Yaskawa INFORM job: X2_34-37(-90,0).JBI

/JOB
//NAME X2_34-37(-90,0)
//POS
///NPOS 478,478,478,11,0,0
///TOOL 0
///POSTYPE PULSE
///PULSE
C00000=59350,-53311,-57323,3430,41392,19515
C00001=122728,-72765,-37270,-45372,18157,11336
C00002=113002,-9355,-31874,-9491,78881,-10162
C00003=107008,40287,15446,-7646,74688,-11911
C00004=107149,45804,24218,-7788,72161,-11701
C00005=108392,48192,28010,-10243,72680,-1076
C00006=108392,48392,29954,-10302,71604,-983
C00007=108392,48331,29423,-10286,71896,-1009
C00008=108010,50265,31522,-10186,71551,-1114
C00009=108392,48331,29423,-10286,71896,-1009
C00010=108911,49901,30550,-10443,72076,-8021
C00011=109414,51873,32709,-10619,71831,-7821
C00012=108911,49901,30550,-10443,72076,-8021
C00013=102203,43615,23227,-8248,72569,-10434
C00014=106081,49085,29485,-15378,74997,-2308
C00015=106081,49206,30588,-15419,74401,-2232
C00016=106081,49153,30130,-15402,74647,-2263
C00017=105730,50968,32108,-15326,74307,-2347
C00018=106081,49153,30130,-15402,74647,-2263
C00019=108167,43461,21271,-12324,74506,-6920
C00020=107374,42085,15448,-7738,75637,-11845
C00021=120191,30165,1303,-6226,81332,6626
C00022=119709,34887,8992,-6124,79003,6581
C00023=119523,36874,12198,-6088,78043,6565
C00024=119519,36825,13807,-6108,77033,6613
C00025=119523,36874,12198,-6088,78043,6565
C00026=119515,36764,13496,-6103,77191,6604
C00027=119868,39633,16467,-6214,76866,6741
C00028=119515,36764,13496,-6103,77191,6604
C00029=121889,32783,9008,-6775,78090,7366
C00030=122776,40716,17165,-7052,77228,7717
C00031=121823,41691,18182,-6780,77023,7402
C00032=122776,40716,17165,-7052,77228,7717
C00033=121889,32783,9008,-6775,78090,7366
C00034=119523,36874,12198,-6088,78043,6565
C00035=119709,34887,8992,-6124,79003,6581
C00036=120191,30165,1303,-6226,81332,6626
C00037=121604,30205,1144,-6630,81559,7083
C00038=121089,34887,8794,-6520,79231,7034
C00039=120890,36858,11983,-6481,78271,7017
C00040=120886,36803,13585,-6502,77262,7069
C00041=120890,36858,11983,-6481,78271,7017
C00042=120878,36774,13282,-6496,77432,7057
C00043=121214,39658,16269,-6601,77105,7189
C00044=120878,36774,13282,-6496,77432,7057
C00045=120486,37076,13561,-6383,77385,6926
C00046=119528,38122,14634,-6107,77190,6608
C00047=120486,37076,13561,-6383,77385,6926
C00048=120682,35058,10322,-6419,78351,6942
C00049=121186,30266,2562,-6523,80690,6990
C00050=134026,40869,15057,4047,52311,47824
C00051=133273,45805,23219,4742,49872,47398
C00052=132981,47914,26662,5033,48858,47219
C00053=132978,48047,28467,5116,47820,47163
C00054=132981,47914,26662,5033,48858,47219
C00055=130421,47335,28194,14259,47961,42182
C00056=130639,50701,31849,14213,47420,42201
C00057=132969,48064,28169,5108,48012,47169
C00058=135543,46606,26609,3148,48091,48321
C00059=135868,54135,34684,2953,46980,48432
C00060=134925,54643,35244,3684,46935,48001
C00061=135868,54135,34684,2953,46980,48432
C00062=135543,46606,26609,3148,48091,48321
C00063=132981,47914,26662,5033,48858,47219
C00064=133273,45805,23219,4742,49872,47398
C00065=134026,40869,15057,4047,52311,47824
C00066=158164,35728,9631,-12841,54320,57618
C00067=156933,39530,16487,-12369,51918,57402
C00068=156452,41160,19364,-12190,50934,57317
C00069=156450,41229,21096,-12367,49926,57444
C00070=156452,41160,19364,-12190,50934,57317
C00071=156479,41102,20610,-12346,50159,57426
C00072=156356,44237,23924,-12335,49721,57428
C00073=156479,41102,20610,-12346,50159,57426
C00074=155785,40986,20547,-11858,50036,57137
C00075=154785,40646,20189,-11137,49940,56708
C00076=155785,40986,20547,-11858,50036,57137
C00077=156262,39303,17617,-12037,51024,57224
C00078=157483,35375,10637,-12509,53434,57446
C00079=160593,39475,13550,-14508,54241,58615
C00080=159342,43270,20469,-14089,51785,58436
C00081=158853,44905,23381,-13934,50776,58367
C00082=158852,45007,25149,-14138,49770,58512
C00083=158853,44905,23381,-13934,50776,58367
C00084=155515,42876,22536,-2607,48655,51694
C00085=155529,45453,25272,-2635,48295,51710
C00086=158854,44932,24718,-14094,49990,58481
C00087=161444,46441,26342,-15939,50249,59595
C00088=161040,53766,34331,-15923,49060,59612
C00089=160097,53171,33669,-15238,48978,59196
C00090=161040,53766,34331,-15923,49060,59612
C00091=161444,46441,26342,-15939,50249,59595
C00092=158853,44905,23381,-13934,50776,58367
C00093=159342,43270,20469,-14089,51785,58436
C00094=160593,39475,13550,-14508,54241,58615
C00095=148971,42504,16746,-4915,52183,53021
C00096=147979,47046,24523,-4355,49683,52716
C00097=147593,48996,27807,-4132,48646,52593
C00098=147590,49137,29621,-4197,47605,52637
C00099=147593,48996,27807,-4132,48646,52593
C00100=148206,49324,28699,-4616,48299,52880
C00101=148386,52346,32006,-4787,47830,52984
C00102=147610,49163,29309,-4198,47810,52637
C00103=147454,49128,29272,-4080,47808,52567
C00104=147457,49325,29466,-4083,47790,52569
C00105=146486,49526,29681,-3347,47716,52137
C00106=147457,49325,29466,-4083,47790,52569
C00107=147454,49128,29272,-4080,47808,52567
C00108=147593,48996,27807,-4132,48646,52593
C00109=147979,47046,24523,-4355,49683,52716
C00110=148753,37651,9035,-4624,54413,52827
C00111=162629,67371,16666,-14387,95994,52782
C00112=162715,57365,2812,-16324,103951,51832
C00113=160874,53905,-839,-17120,106140,50911
C00114=173545,40340,-5560,-32046,95660,52318
C00115=172356,48440,2674,-29251,92100,53433
C00116=172375,50726,4522,-29031,92137,53493
C00117=171941,50016,3368,-28017,91820,53556
C00118=172934,47472,3029,-30290,87254,54349
C00119=166298,46940,-5204,-15814,93409,53604
C00120=167727,47900,-7727,-16302,95626,53755
C00121=154370,-11928,-49618,9666,90717,31299
C00122=126601,-55902,-47749,13735,83134,-9694
C00123=110572,-56965,-55890,14658,90278,-14468
C00124=134387,-39172,-38807,-12376,86277,20344
C00125=136266,-41846,-34601,-16059,78566,27361
C00126=135831,-39745,-32201,-16023,78101,27269
C00127=132382,-45209,-35546,-15612,76705,26216
C00128=133414,-53213,-38184,-18925,70500,23054
C00129=132483,-55031,-38922,-19056,69495,22520
C00130=133928,-49591,-35946,-21097,73532,26608
C00131=127522,-56914,-39892,-20235,70668,24713
C00132=130575,-58808,-42172,-20683,71834,25657
C00133=131419,-52897,-41760,-13173,72105,2236
C00134=151757,-37235,-32664,-25855,92713,16023
C00135=148694,-31120,-30848,-28555,97484,16481
C00136=152363,20888,-11521,-23566,108052,25705
C00137=155491,63274,13853,-18429,111086,34801
C00138=150514,89045,46229,-21307,107758,32982
C00139=149106,88504,48693,-21100,105732,32842
C00140=153713,50743,12699,-33613,93756,12076
C00141=152514,62453,23514,-30409,96198,11306
C00142=153571,72354,35346,-30285,92331,9677
C00143=151039,57679,18624,-26133,86933,-1110
C00144=146574,45095,4989,-17377,80841,-11651
C00145=146416,46512,5286,-14277,82040,-14909
C00146=141388,39329,-953,-2943,76634,-26635
C00147=140619,46287,2526,-1728,82676,-28626
C00148=139837,43342,-3801,-1439,85041,-28899
C00149=141798,27002,-27786,-2149,91441,-28405
C00150=143772,-19107,-38740,-14355,94017,12677
C00151=143698,-35148,-33847,-20276,92427,33189
C00152=141918,-24797,-26817,-20326,92921,32464
C00153=139594,-23350,-22642,-20301,90627,32011
C00154=140500,-47178,-33366,-23894,71804,30939
C00155=143725,-38410,-27629,-28409,78422,12628
C00156=143636,-41247,-28872,-28024,73501,10134
C00157=137881,-52583,-35183,-23334,62436,-881
C00158=129248,-60396,-38780,-13341,52739,-14402
C00159=124267,-62494,-40095,-3055,50610,-24451
C00160=119084,-58248,-39599,7242,55598,-36917
C00161=117935,-60108,-42034,7672,56240,-37337
C00162=115664,-65010,-47736,8512,57449,-38158
C00163=121785,-61828,-52329,5505,69210,-35118
C00164=148930,-33628,-41038,-4538,77484,-18447
C00165=163858,24222,1645,-10794,81228,-7547
C00166=163712,28964,9442,-10824,78886,-7392
C00167=163375,31110,12798,-10770,77896,-7422
C00168=162966,25989,8902,-6453,74358,251
C00169=171220,35624,19743,-19386,77626,18928
C00170=174903,69588,56637,-24731,86432,36485
C00171=176281,62245,51753,-30189,71814,61901
C00172=174700,53660,39403,-25265,70725,61619
C00173=176244,52382,34806,-25393,73168,61673
C00174=174832,57379,31343,-14926,87681,59388
C00175=147451,1111,-29714,-5377,100632,19781
C00176=112791,-31989,-50015,2241,90212,-24459
C00177=107981,-35875,-46971,4517,78040,-26268
C00178=109410,-31915,-41181,4141,76439,-25836
C00179=109643,-29612,-38300,4087,75838,-25775
C00180=108775,-25319,-36143,8282,81258,-19579
C00181=113815,-28658,-38499,3030,79667,-8408
C00182=120146,-28725,-38561,-4150,79807,1674
C00183=136607,-12516,-23650,-24736,88445,21917
C00184=138997,-10914,-21244,-25939,84896,23287
C00185=136597,-19153,-27062,-20495,74929,32505
C00186=127631,-24253,-35023,-5775,74490,30240
C00187=129181,-27934,-40726,-6212,76213,30690
C00188=139651,-3107,-33687,-4364,86662,-15844
C00189=140099,618,-27389,-4493,84729,-15631
C00190=139833,2398,-24483,-4425,83841,-15689
C00191=138545,5945,-22338,1327,87046,-9478
C00192=148216,2445,-23282,-11424,83992,10224
C00193=153040,10099,-16158,-17812,86817,20381
C00194=156294,19571,-6705,-22682,89726,28901
C00195=159272,37595,11787,-27323,93895,28698
C00196=154169,16276,-8816,-16740,78788,38767
C00197=152712,20066,-9195,-12847,84122,38020
C00198=154297,18366,-13942,-13242,86364,38311
C00199=143466,6998,19042,-5158,32162,41222
C00200=147237,-51968,-50099,4175,73083,42408
C00201=-3643,-76224,-106676,-19950,71810,-76872
C00202=-6047,-95755,-92046,14751,98253,-9605
C00203=-2299,-70459,-84112,3705,91093,-18065
C00204=-2299,-70459,-84112,3705,91093,-18065
C00205=-2299,-70459,-84112,3705,91093,-18065
C00206=-2299,-70459,-84112,3705,91093,-18065
C00207=61951,-108908,-90353,7974,21769,-53190
C00208=44975,-75191,-76287,54105,62461,-71292
C00209=78581,-58710,-61930,31634,35162,-55381
C00210=94816,-22771,-39143,38147,43253,-85351
C00211=95668,-20492,-32997,40754,37729,-87628
C00212=95668,-20442,-31356,41600,36978,-88107
C00213=95668,-20481,-32513,41001,37505,-87770
C00214=95495,-18068,-30743,41020,37699,-87770
C00215=95668,-20481,-32513,41001,37505,-87770
C00216=89708,-21268,-34265,45191,40885,-89740
C00217=90261,-15540,-28471,45297,40161,-89843
C00218=90261,-15513,-27582,45749,39780,-90110
C00219=90261,-15527,-28007,45532,39961,-89983
C00220=91375,-15045,-27644,44668,39419,-89560
C00221=90261,-15527,-28007,45532,39961,-89983
C00222=88067,4046,-12693,46606,41526,-90451
C00223=88067,4066,-11724,47089,41117,-90741
C00224=88067,4053,-12277,46812,41349,-90575
C00225=89178,4455,-11933,46018,40776,-90188
C00226=88067,4046,-12908,46498,41617,-90387
C00227=93864,-1171,-17172,27469,32670,-81316
C00228=93864,-1150,-16127,27931,32107,-81561
C00229=93864,-1161,-16600,27720,32361,-81450
C00230=93686,724,-15030,27925,32421,-81546
C00231=93864,-1171,-17458,27343,32827,-81250
C00232=86880,-2670,-19039,34652,35541,-84684
C00233=77447,40941,12142,46518,66528,-79108
C00234=77447,40828,13235,46743,66015,-79371
C00235=77447,40915,12396,46570,66408,-79170
C00236=78189,41279,12776,46293,66002,-79003
C00237=77447,40915,12396,46570,66408,-79170
C00238=77711,61383,34518,44784,60703,-78470
C00239=77711,61401,35861,45103,60114,-78770
C00240=77711,61383,34367,44748,60769,-78437
C00241=78627,62334,35456,44423,60182,-78251
C00242=77711,61383,34367,44748,60769,-78437
C00243=87327,38488,-37,11684,57539,-57739
C00244=92703,33891,441,-7168,52274,-42102
C00245=94252,42993,11540,-8600,52099,-41498
C00246=94252,42798,12742,-8697,51267,-41425
C00247=94252,42977,11640,-8607,52029,-41490
C00248=94205,45159,13958,-8608,51725,-41483
C00249=94252,42977,11640,-8607,52029,-41490
C00250=88553,40317,7447,-4237,52798,-43866
C00251=77780,64504,35767,30085,55551,-63063
C00252=77882,64751,36053,30043,55472,-63041
C00253=77882,64734,37138,30274,54883,-63228
C00254=77882,64751,36157,30064,55416,-63059
C00255=78504,65403,36908,29747,55085,-62879
C00256=77882,64751,36157,30064,55416,-63059
C00257=77930,65478,35918,25842,53172,-64425
C00258=75957,78225,52136,32216,53612,-64557
C00259=75957,78336,53316,32477,53042,-64758
C00260=75957,78231,52217,32233,53572,-64572
C00261=76543,78457,52489,31920,53306,-64380
C00262=75957,78231,52217,32233,53572,-64572
C00263=75783,52857,14963,26033,68951,-61065
C00264=76778,51540,16645,25850,67104,-61119
C00265=76553,54259,19675,26040,66751,-61289
C00266=76152,68337,35819,26754,64443,-62008
C00267=76309,68979,36633,26729,64087,-61973
C00268=76161,73805,46213,28343,55084,-61966
C00269=76040,75497,47702,28425,55082,-62022
C00270=75485,77195,52229,31394,50715,-63899
C00271=76358,61277,29656,23751,52989,-59172
C00272=75244,23807,-9833,23130,57943,-58480
C00273=78328,30150,-3634,21247,56637,-57509
C00274=82524,40429,3879,10756,62616,-55403
C00275=83243,40821,5102,10290,61963,-55146
C00276=92066,29463,-1741,-9440,53850,-44784
C00277=92409,29931,-1279,-9693,53846,-44645
C00278=95822,30058,-1154,-12140,54276,-43316
C00279=92072,29548,-1666,-1163,53131,-49252
C00280=90114,17633,-16179,284,55928,-50028
C00281=80680,14818,-24193,20442,65844,-59872
C00282=77180,38928,7111,43331,74666,-71993
C00283=76673,54469,24090,43953,73098,-72919
C00284=76771,55672,25429,43962,72900,-72963
C00285=76784,55849,25626,43964,72871,-72969
C00286=78172,63512,34338,39520,65661,-69940
C00287=79648,59091,29288,35397,62522,-67074
C00288=75980,37060,-454,35377,69732,-66149
C00289=81483,21043,-13915,32107,67437,-64274
C00290=93507,15990,-19907,5211,64480,-50669
C00291=99800,11020,-22513,-5623,60000,-50039
C00292=99783,5101,-23986,-5176,53212,-49502
C00293=100096,6075,-23185,433,53012,-52451
C00294=100559,6099,-23054,81,52942,-52266
C00295=100559,6099,-23054,81,52942,-52266
C00296=95780,-7481,-38206,3595,55393,-54089
C00297=86068,-7258,-38029,32714,65078,-69570
C00298=89977,-5445,-32844,31222,61873,-68759
C00299=89643,-3500,-31211,31407,61985,-68864
C00300=88246,9256,-20330,32202,62368,-69333
C00301=88278,10099,-19644,32183,62365,-69319
C00302=87437,19709,-10754,32777,62224,-69720
C00303=93562,10508,-19170,18010,55559,-61503
C00304=91617,5056,-25544,19093,57043,-62018
C00305=90732,-18366,-45622,16723,54511,-62954
C00306=99990,-18392,-38429,13920,44377,-71620
C00307=100837,-18665,-38703,13148,44269,-71234
C00308=97918,-19792,-36092,25968,40989,-77255
C00309=98001,-23338,-34358,32939,34367,-85184
C00310=99551,-14617,-34520,26965,45535,-82533
C00311=93873,-14551,-28302,47146,43784,-90863
C00312=93873,-14551,-28302,47146,43784,-90863
C00313=92894,-25654,-38538,40707,40207,-87648
C00314=51114,-81290,-74278,61960,52593,-60278
C00315=6076,-109546,-85200,71251,79672,-70600
C00316=6076,-109546,-85200,71251,79672,-70600
C00317=6076,-109546,-85200,-4239,76823,-70600
C00318=-8024,-164446,-133802,16041,6272,-12396
C00319=-8024,-164446,-133802,16041,6272,-12396
C00320=-80911,-131071,-112390,19160,57527,4768
C00321=-107387,-112645,-89313,18613,48039,3448
C00322=-120529,-94925,-67119,18087,38914,2179
C00323=-102807,-11704,-32462,5874,76695,13415
C00324=-103436,-3791,-23255,6127,75148,13126
C00325=-103560,-1765,-20423,6188,74460,13051
C00326=-103560,-1806,-19122,6212,73642,13010
C00327=-103601,-1431,-19452,6214,74041,13015
C00328=-104452,277,-18031,6506,74110,12725
C00329=-103539,-2063,-20212,6189,74177,13043
C00330=-120126,-10436,-31938,6011,80471,-6680
C00331=-119034,-8056,-29018,5697,79822,-6345
C00332=-119034,-8150,-28117,5707,79221,-6375
C00333=-119034,-8056,-29018,5697,79822,-6345
C00334=-118636,-7203,-28340,5579,79816,-6211
C00335=-119064,-5644,-27091,5704,79877,-6351
C00336=-118636,-7203,-28340,5579,79816,-6211
C00337=-122253,-9472,-30321,6643,80135,-7408
C00338=-122707,-3013,-24427,6779,79866,-7571
C00339=-122021,-2022,-23613,6578,79819,-7343
C00340=-122707,-3013,-24427,6779,79866,-7571
C00341=-121204,9301,-16198,6319,81003,-7011
C00342=-120979,11415,-12534,6272,79823,-6996
C00343=-120979,11346,-11871,6278,79382,-7018
C00344=-120979,11415,-12534,6272,79823,-6996
C00345=-121673,13624,-10544,6477,79786,-7230
C00346=-120979,11415,-12534,6272,79823,-6996
C00347=-121039,12182,-11846,8037,80321,-9006
C00348=-120294,13253,-10880,7825,80206,-8763
C00349=-121039,12182,-11846,8037,80321,-9006
C00350=-121310,5674,-20943,6336,82061,-6993
C00351=-139815,-25323,-43479,19,53677,-50237
C00352=-137572,-18164,-33682,-1617,51348,-49297
C00353=-137572,-18186,-32944,-1627,50884,-49290
C00354=-137572,-18164,-33682,-1617,51348,-49297
C00355=-138000,-16627,-32540,-1306,51428,-49477
C00356=-137572,-18164,-33682,-1617,51348,-49297
C00357=-141541,-18207,-34048,1274,51544,-50959
C00358=-141186,-12326,-28968,1018,51433,-50811
C00359=-140737,-11536,-28358,690,51458,-50623
C00360=-141186,-12326,-28968,1018,51433,-50811
C00361=-159686,26179,2441,14066,53601,-58348
C00362=-159232,27229,5186,13963,52408,-58323
C00363=-159232,27222,5932,14048,51958,-58386
C00364=-159232,27229,5186,13963,52408,-58323
C00365=-159232,27225,5485,13997,52227,-58349
C00366=-159220,29212,7438,14024,52052,-58369
C00367=-159232,27225,5485,13997,52227,-58349
C00368=-164735,35698,13654,29808,58437,-68077
C00369=-164028,35618,13572,29436,58200,-67836
C00370=-164735,35698,13654,29808,58437,-68077
C00371=-161795,29787,7764,15728,52595,-59373
C00372=-161795,29788,8601,15834,52098,-59452
C00373=-161795,29787,7764,15728,52595,-59373
C00374=-161783,31729,9695,15761,52409,-59396
C00375=-161795,29787,7764,15728,52595,-59373
C00376=-165243,28841,7606,18106,52930,-60800
C00377=-165806,38731,16984,22046,53706,-63214
C00378=-165192,38605,16853,21659,53559,-62976
C00379=-165806,38731,16984,22046,53706,-63214
C00380=-161708,46386,23154,8907,61269,-44547
C00381=-161224,48066,26131,8737,60259,-44442
C00382=-161222,48202,27939,8826,59228,-44523
C00383=-161224,48066,26131,8737,60259,-44442
C00384=-161238,48238,27638,8816,59431,-44513
C00385=-161118,51495,31180,8798,58918,-44508
C00386=-161238,48238,27638,8816,59431,-44513
C00387=-161086,48113,27502,8735,59433,-44454
C00388=-161078,48307,27691,8732,59416,-44452
C00389=-160108,47930,27281,8216,59373,-44078
C00390=-161078,48307,27691,8732,59416,-44452
C00391=-161086,48113,27502,8735,59433,-44454
C00392=-161224,48066,26131,8737,60259,-44442
C00393=-161708,46386,23154,8907,61269,-44547
C00394=-162944,42495,16096,9351,63722,-44812
C00395=-174609,85782,55206,18480,94121,-57514
C00396=-173388,84153,56528,18357,92279,-57362
C00397=-178295,72858,49572,29598,87914,-53870
C00398=-178363,71681,49458,30316,81279,-55416
C00399=-178775,74747,53745,31442,79609,-55982
C00400=-178120,80280,53499,25679,87195,-54196
C00401=-177788,66292,45128,22799,80541,-57078
C00402=-165876,20944,-7359,14016,91072,-47752
C00403=-144031,-8096,-47002,-481,102749,-33013
C00404=-113249,-55125,-55779,-6617,87879,14622
C00405=-105402,-49476,-43093,-17129,78821,17705
C00406=-107372,-45114,-37354,-16923,77172,17229
C00407=-107897,-43226,-34630,-16890,76385,17150
C00408=-123036,-54169,-41018,3647,66196,9526
C00409=-125103,-54109,-40569,7539,65613,9158
C00410=-133018,-52183,-38196,18552,67287,3963
C00411=-135096,-56008,-41994,19101,68310,3149
C00412=-148619,-36280,-33179,26254,90102,-11601
C00413=-132022,-46525,-51369,8915,93592,-12104
C00414=-152394,4325,-31091,21424,100011,-27739
C00415=-150620,74441,30669,21497,109248,-32750
C00416=-152126,53419,9650,25324,101365,-34081
C00417=-152823,56464,14992,29675,98105,-11003
C00418=-153512,66710,26766,28901,94570,-8735
C00419=-151176,53481,12027,24882,88967,903
C00420=-148217,46273,4019,19056,85273,8690
C00421=-145575,40234,-2364,10924,81880,17637
C00422=-142774,42237,-1321,4504,82417,25550
C00423=-141310,41249,-3509,1904,83312,28397
C00424=-140520,38377,-9680,1608,85617,28672
C00425=-145482,-30493,-50756,14636,95383,-13188
C00426=-142176,-26033,-28146,20229,92686,-32606
C00427=-139838,-24569,-23969,20194,90398,-32145
C00428=-141333,-43488,-32424,24355,75177,-35516
C00429=-142946,-39788,-29545,27566,77515,-12382
C00430=-142712,-38988,-29426,26650,76094,-9122
C00431=-137490,-51139,-36024,22440,64589,1384
C00432=-129219,-61272,-40095,12800,52551,14455
C00433=-125098,-62268,-41395,3949,52110,22670
C00434=-120434,-59895,-41306,-5152,54802,34175
C00435=-118218,-60267,-42467,-7826,55944,37248
C00436=-115940,-65207,-48159,-8687,57132,38075
C00437=-158051,-33814,-49892,7441,80913,13725
C00438=-163513,25616,3177,10792,80459,7597
C00439=-163372,30455,11081,10830,78103,7439
C00440=-163993,28142,11085,12803,74423,6981
C00441=-161648,29238,11147,4496,75447,179
C00442=-171143,45412,28292,19077,81279,-23270
C00443=-173705,65046,50293,22854,85176,-36170
C00444=-173974,62485,49606,24076,73199,-49227
C00445=-172570,70781,55370,19160,78152,-47867
C00446=-174025,68948,50025,19270,80716,-47984
C00447=-170072,38309,9009,5458,81396,-48416
C00448=-145937,-33300,-50613,2555,87892,-10434
C00449=-117969,-26674,-50251,-1455,96093,22658
C00450=-108065,-36096,-47601,-4778,77881,26213
C00451=-109507,-32110,-41823,-4391,76297,25779
C00452=-109013,-37865,-42571,-5415,69231,26193
C00453=-107679,-33877,-40967,-9851,74714,20356
C00454=-113110,-32097,-41032,-3661,77261,8676
C00455=-119719,-29513,-40298,3828,79988,-1546
C00456=-130402,-22376,-34110,15555,82843,-20591
C00457=-132503,-6978,-23545,15597,88653,-21115
C00458=-133170,-4219,-21374,15691,88857,-21320
C00459=-127848,-25408,-36231,5685,74178,-30350
C00460=-129407,-29126,-41925,6135,75876,-30806
C00461=-139811,-3516,-34603,4319,86523,15767
C00462=-140259,233,-28314,4452,84609,15556
C00463=-139695,2013,-26001,4296,84073,15716
C00464=-138357,5152,-24179,-1260,87195,9766
C00465=-142581,5884,-23661,3711,87904,-1101
C00466=-150814,13438,-16434,14780,91136,-16214
C00467=-153585,30594,-714,18230,97958,-27100
C00468=-154794,42503,11376,18274,96962,-27667
C00469=-154809,42525,11398,18275,96963,-27672
C00470=-153093,18834,-10833,12947,84050,-38162
C00471=-154693,17143,-15552,13354,86281,-38457
C00472=-149017,-30265,-44675,21897,62232,-30468
C00473=-102406,-109115,-77602,2898,35707,11807
C00474=-80911,-131071,-112390,19160,57527,4768
C00475=-8024,-164446,-133802,16041,6272,-12396
C00476=-8024,-164446,-133802,16041,6272,-12396
C00477=6076,-109546,-85200,-4239,76823,-70600
BC00000=228604,517006,641220
BC00001=287751,517515,392862
BC00002=287751,487719,199707
BC00003=287751,487719,199707
BC00004=287751,487719,199707
BC00005=287751,487719,199707
BC00006=287751,487719,199707
BC00007=287751,487719,199707
BC00008=287751,487719,199707
BC00009=287751,487719,199707
BC00010=287751,487719,199707
BC00011=287751,487719,199707
BC00012=287751,487719,199707
BC00013=287751,487719,199707
BC00014=287751,487719,199707
BC00015=287751,487719,199707
BC00016=287751,487719,199707
BC00017=287751,487719,199707
BC00018=287751,487719,199707
BC00019=287751,487719,199707
BC00020=287751,487719,199707
BC00021=325450,480985,183037
BC00022=325450,480985,183037
BC00023=325450,480985,183037
BC00024=325450,480985,183037
BC00025=325450,480985,183037
BC00026=325450,480985,183037
BC00027=325450,480985,183037
BC00028=325450,480985,183037
BC00029=325450,480985,183037
BC00030=325450,480985,183037
BC00031=325450,480985,183037
BC00032=325450,480985,183037
BC00033=325450,480985,183037
BC00034=325450,480985,183037
BC00035=325450,480985,183037
BC00036=325450,480985,183037
BC00037=304393,460388,181316
BC00038=304393,460388,181316
BC00039=304393,460388,181316
BC00040=304393,460388,181316
BC00041=304393,460388,181316
BC00042=304393,460388,181316
BC00043=304393,460388,181316
BC00044=304393,460388,181316
BC00045=304393,460388,181316
BC00046=304393,460388,181316
BC00047=304393,460388,181316
BC00048=304393,460388,181316
BC00049=304393,460388,181316
BC00050=360925,503974,119018
BC00051=360925,503974,119018
BC00052=360925,503974,119018
BC00053=360925,503974,119018
BC00054=360925,503974,119018
BC00055=360925,503974,119018
BC00056=360925,503974,119018
BC00057=360925,503974,119018
BC00058=360925,503974,119018
BC00059=360925,503974,119018
BC00060=360925,503974,119018
BC00061=360925,503974,119018
BC00062=360925,503974,119018
BC00063=360925,503974,119018
BC00064=360925,503974,119018
BC00065=360925,503974,119018
BC00066=398158,448100,117989
BC00067=398158,448100,117989
BC00068=398158,448100,117989
BC00069=398158,448100,117989
BC00070=398158,448100,117989
BC00071=398158,448100,117989
BC00072=398158,448100,117989
BC00073=398158,448100,117989
BC00074=398158,448100,117989
BC00075=398158,448100,117989
BC00076=398158,448100,117989
BC00077=398158,448100,117989
BC00078=398158,448100,117989
BC00079=397418,451841,118275
BC00080=397418,451841,118275
BC00081=397418,451841,118275
BC00082=397418,451841,118275
BC00083=397418,451841,118275
BC00084=397418,451841,118275
BC00085=397418,451841,118275
BC00086=397418,451841,118275
BC00087=397418,451841,118275
BC00088=397418,451841,118275
BC00089=397418,451841,118275
BC00090=397418,451841,118275
BC00091=397418,451841,118275
BC00092=397418,451841,118275
BC00093=397418,451841,118275
BC00094=397418,451841,118275
BC00095=337741,442196,121007
BC00096=337741,442196,121007
BC00097=337741,442196,121007
BC00098=337741,442196,121007
BC00099=337741,442196,121007
BC00100=337741,442196,121007
BC00101=337741,442196,121007
BC00102=337741,442196,121007
BC00103=337741,442196,121007
BC00104=337741,442196,121007
BC00105=337741,442196,121007
BC00106=337741,442196,121007
BC00107=337741,442196,121007
BC00108=337741,442196,121007
BC00109=337741,442196,121007
BC00110=337741,442196,121007
BC00111=362486,406092,31407
BC00112=351094,389162,16365
BC00113=343454,385623,9383
BC00114=366302,380877,17
BC00115=366302,380877,17
BC00116=366302,380877,17
BC00117=366302,380877,17
BC00118=366302,380877,17
BC00119=366302,380877,17
BC00120=366302,380877,17
BC00121=351235,377860,125844
BC00122=328122,373227,305595
BC00123=350132,373227,305595
BC00124=350701,373152,305427
BC00125=350701,373152,305427
BC00126=350701,373152,305427
BC00127=350701,373152,305427
BC00128=350701,373152,305423
BC00129=350699,373153,305422
BC00130=350701,373152,305423
BC00131=350701,373152,305423
BC00132=350701,373152,305423
BC00133=350701,373152,305427
BC00134=350701,373152,305427
BC00135=350132,373227,305595
BC00136=357470,406535,171187
BC00137=363729,434945,56545
BC00138=350092,440820,42081
BC00139=350092,440820,42081
BC00140=350092,440820,42081
BC00141=350092,440820,42081
BC00142=350092,440820,42081
BC00143=350092,440820,42081
BC00144=350092,440820,42081
BC00145=350092,440820,42081
BC00146=350092,440820,42081
BC00147=350092,440820,42081
BC00148=350092,440820,42081
BC00149=350029,441190,44115
BC00150=332813,387958,218553
BC00151=324205,361343,305772
BC00152=324267,360974,303737
BC00153=324267,360974,303737
BC00154=324267,360974,303737
BC00155=324267,360974,303737
BC00156=324267,360974,303737
BC00157=324267,360974,303737
BC00158=324267,360974,303737
BC00159=324267,360974,303737
BC00160=324267,360974,303737
BC00161=324267,360974,303737
BC00162=324267,360974,303737
BC00163=324205,361343,305772
BC00164=365888,380957,256640
BC00165=398158,394894,219979
BC00166=398158,394894,219979
BC00167=398158,394894,219979
BC00168=398158,394894,219979
BC00169=398158,394894,219979
BC00170=398158,394894,219979
BC00171=398158,394894,219979
BC00172=398158,394894,219979
BC00173=398158,394894,219979
BC00174=398158,394894,219979
BC00175=365105,398728,219938
BC00176=328853,402933,219893
BC00177=328853,402933,219893
BC00178=328853,402933,219893
BC00179=328853,402933,219893
BC00180=328853,402933,219893
BC00181=328853,402933,219893
BC00182=328853,402933,219893
BC00183=328853,402933,219893
BC00184=328853,402933,219893
BC00185=328853,402933,219893
BC00186=328853,402933,219893
BC00187=328853,402933,219893
BC00188=366727,414928,149826
BC00189=366727,414928,149826
BC00190=366727,414928,149826
BC00191=366727,414928,149826
BC00192=366727,414928,149826
BC00193=366727,414928,149826
BC00194=366727,414928,149826
BC00195=366727,414928,149826
BC00196=366727,414928,149826
BC00197=366727,414928,149826
BC00198=366727,414928,149826
BC00199=366727,515070,355741
BC00200=366727,515070,355741
BC00201=199448,515539,1075137
BC00202=95028,515070,919110
BC00203=123826,515279,972180
BC00204=123826,515279,972180
BC00205=123826,515279,972180
BC00206=44761,462630,27794
BC00207=44761,462630,27794
BC00208=44761,462630,27793
BC00209=44761,462630,27793
BC00210=44761,462630,27793
BC00211=44761,462631,27793
BC00212=44761,462631,27793
BC00213=44761,462631,27793
BC00214=44761,462631,27793
BC00215=44761,462631,27793
BC00216=44761,462631,27793
BC00217=44761,462631,27793
BC00218=44761,462631,27793
BC00219=44761,462631,27793
BC00220=44761,462631,27793
BC00221=44761,462631,27793
BC00222=44761,462631,27793
BC00223=44761,462631,27793
BC00224=44761,462631,27793
BC00225=44761,462631,27793
BC00226=44761,462631,27793
BC00227=44761,462631,27793
BC00228=44761,462631,27793
BC00229=44761,462631,27793
BC00230=44761,462631,27793
BC00231=44761,462631,27793
BC00232=44761,462631,27793
BC00233=44761,462631,27793
BC00234=44761,462631,27793
BC00235=44761,462631,27793
BC00236=44761,462631,27793
BC00237=44761,462631,27793
BC00238=44761,462631,27793
BC00239=44761,462631,27793
BC00240=44761,462631,27793
BC00241=44761,462631,27793
BC00242=44761,462631,27793
BC00243=44761,462631,27793
BC00244=44761,462630,27793
BC00245=44761,462630,27793
BC00246=44761,462630,27793
BC00247=44761,462630,27793
BC00248=44761,462630,27793
BC00249=44761,462630,27793
BC00250=44761,462630,27793
BC00251=44761,462630,27793
BC00252=44761,462630,27793
BC00253=44761,462630,27793
BC00254=44761,462630,27793
BC00255=44761,462630,27793
BC00256=44761,462630,27793
BC00257=44761,453221,27793
BC00258=44761,453221,27793
BC00259=44761,453221,27793
BC00260=44761,453221,27793
BC00261=44761,453221,27793
BC00262=44761,453221,27793
BC00263=45255,444613,27793
BC00264=45255,444613,27793
BC00265=45255,444613,27793
BC00266=45255,444613,27793
BC00267=45255,444613,27793
BC00268=45255,444613,27793
BC00269=45255,444613,27793
BC00270=45255,444613,27793
BC00271=45255,444613,27793
BC00272=45255,444613,27793
BC00273=45255,444613,27793
BC00274=45255,444613,27793
BC00275=45253,444683,27793
BC00276=45253,444683,27793
BC00277=45253,444683,27793
BC00278=45253,444683,27793
BC00279=45253,444683,27793
BC00280=45253,444683,27793
BC00281=44971,454975,27792
BC00282=44971,454975,27792
BC00283=44971,454975,27792
BC00284=44971,454975,27792
BC00285=44971,454975,27792
BC00286=44970,454994,27792
BC00287=44970,454994,27792
BC00288=44970,454994,27792
BC00289=44966,455154,27792
BC00290=44966,455154,27792
BC00291=44966,455154,27792
BC00292=44966,455154,27792
BC00293=44966,455154,27792
BC00294=44966,455154,27792
BC00295=44966,455154,27792
BC00296=44966,455154,27792
BC00297=44966,455154,27792
BC00298=44957,455470,27792
BC00299=44957,455470,27792
BC00300=44957,455470,27792
BC00301=44957,455470,27792
BC00302=44957,455470,27792
BC00303=44957,455470,27792
BC00304=44957,455470,27792
BC00305=44859,459040,27792
BC00306=44823,460358,27792
BC00307=44823,460358,27792
BC00308=44823,460358,27792
BC00309=44823,460358,27792
BC00310=44823,460358,27792
BC00311=44823,460358,27792
BC00312=44823,460358,27792
BC00313=44823,460358,27792
BC00314=44761,462630,27793
BC00315=44761,546100,27793
BC00316=44761,546100,27793
BC00317=44761,546100,971290
BC00318=95028,515070,1075193
BC00319=235797,-155466,1075193
BC00320=291717,-173504,501205
BC00321=295026,-175720,344845
BC00322=288092,-177851,194471
BC00323=288092,-175723,194471
BC00324=288092,-179084,194471
BC00325=288092,-179155,194471
BC00326=288092,-179155,194471
BC00327=288092,-179505,194471
BC00328=288092,-179505,194471
BC00329=288092,-178804,194471
BC00330=325818,-178589,177096
BC00331=325818,-177793,177096
BC00332=325818,-177793,177096
BC00333=325818,-177793,177096
BC00334=325818,-177793,177096
BC00335=325818,-177793,177096
BC00336=325818,-177793,177096
BC00337=325818,-178114,177096
BC00338=325818,-178659,177096
BC00339=325818,-178659,177096
BC00340=325818,-178659,177096
BC00341=304782,-177778,175837
BC00342=304782,-178169,175837
BC00343=304782,-178169,175837
BC00344=304782,-178169,175837
BC00345=304782,-178169,175837
BC00346=304782,-178169,175837
BC00347=304782,-178169,175837
BC00348=304782,-178169,175837
BC00349=304782,-178169,175837
BC00350=304782,-178605,175837
BC00351=360300,-177931,111224
BC00352=360300,-177638,111224
BC00353=360300,-177638,111224
BC00354=360300,-177638,111224
BC00355=360300,-177638,111224
BC00356=360300,-177638,111224
BC00357=360300,-178156,111224
BC00358=360300,-177428,111224
BC00359=360300,-177428,111224
BC00360=360300,-177428,111224
BC00361=398158,-177653,110801
BC00362=398158,-175808,110801
BC00363=398158,-175808,110801
BC00364=398158,-175808,110801
BC00365=398158,-175808,110801
BC00366=398158,-175808,110801
BC00367=398158,-175808,110801
BC00368=398158,-175808,110801
BC00369=398158,-175808,110801
BC00370=398158,-175808,110801
BC00371=397168,-178328,111236
BC00372=397168,-178328,111236
BC00373=397168,-178328,111236
BC00374=397168,-178328,111236
BC00375=397168,-178328,111236
BC00376=397168,-176350,111236
BC00377=397168,-177173,111236
BC00378=397168,-177173,111236
BC00379=397168,-177173,111236
BC00380=375485,-155755,156312
BC00381=375485,-155755,156312
BC00382=375485,-155755,156312
BC00383=375485,-155755,156312
BC00384=375485,-155755,156312
BC00385=375485,-155755,156312
BC00386=375485,-155755,156312
BC00387=375485,-155755,156312
BC00388=375485,-155755,156312
BC00389=375485,-155755,156312
BC00390=375485,-155755,156312
BC00391=375485,-155755,156312
BC00392=375485,-155755,156312
BC00393=375485,-155755,156312
BC00394=375485,-155755,156312
BC00395=398158,-131674,135077
BC00396=398158,-131674,135077
BC00397=398158,-131674,135077
BC00398=398158,-131674,135077
BC00399=398158,-131674,135077
BC00400=398158,-131674,135074
BC00401=398158,-131674,199522
BC00402=369939,-130367,190529
BC00403=332637,-128291,176238
BC00404=350430,-116776,300608
BC00405=351034,-116702,300430
BC00406=351034,-116702,300430
BC00407=351034,-116702,300430
BC00408=351034,-116702,300430
BC00409=351034,-116702,300430
BC00410=351034,-116702,300430
BC00411=351034,-116702,300430
BC00412=351034,-116702,300430
BC00413=350430,-116776,300608
BC00414=350314,-155460,140475
BC00415=350302,-172845,38361
BC00416=350303,-172143,38359
BC00417=350302,-179079,38361
BC00418=350302,-179079,38361
BC00419=350302,-179079,38361
BC00420=350302,-179079,38357
BC00421=350302,-179079,38361
BC00422=350302,-179079,38361
BC00423=350302,-179079,38361
BC00424=350302,-179079,38361
BC00425=332891,-129402,215544
BC00426=324453,-104426,299301
BC00427=324453,-104426,299301
BC00428=324453,-104426,299301
BC00429=324453,-104426,299301
BC00430=324453,-104426,299301
BC00431=324453,-104426,299301
BC00432=324453,-104426,299301
BC00433=324453,-104426,299301
BC00434=324454,-104427,299300
BC00435=324453,-104426,299301
BC00436=324453,-104426,299301
BC00437=378041,-129317,238802
BC00438=398158,-141033,220588
BC00439=398158,-141033,220588
BC00440=398158,-141033,220588
BC00441=398158,-141033,220588
BC00442=398158,-141033,220588
BC00443=398158,-141033,220588
BC00444=398158,-141033,220588
BC00445=398158,-141033,220588
BC00446=398158,-141033,220588
BC00447=398158,-138511,215353
BC00448=359670,-143049,214660
BC00449=329106,-146653,214110
BC00450=329106,-146653,214110
BC00451=329106,-146653,214110
BC00452=329106,-146653,214110
BC00453=329106,-146653,214110
BC00454=329106,-146653,214110
BC00455=329106,-146653,214110
BC00456=329106,-146653,214110
BC00457=329106,-146653,214110
BC00458=329106,-146653,214110
BC00459=329106,-146653,214110
BC00460=329106,-146653,214110
BC00461=366999,-158610,144660
BC00462=366999,-158610,144660
BC00463=366999,-158610,144660
BC00464=366999,-158610,144660
BC00465=366999,-158610,144660
BC00466=366999,-158610,144660
BC00467=366999,-158610,144660
BC00468=366999,-158610,144660
BC00469=366999,-158610,144660
BC00470=366999,-158610,144660
BC00471=366999,-158610,144660
BC00472=346592,-164721,157542
BC00473=288092,-170050,194471
BC00474=269879,-173504,501205
BC00475=235797,-155466,1075193
BC00476=95028,515070,1075193
BC00477=44761,546100,971290
EC00000=798156,-183832
EC00001=798156,-183832
EC00002=798156,-183832
EC00003=798156,-183832
EC00004=798156,-183832
EC00005=798156,-183832
EC00006=798156,-183832
EC00007=798156,-183832
EC00008=798156,-183832
EC00009=798156,-183832
EC00010=798156,-183832
EC00011=798156,-183832
EC00012=798156,-183832
EC00013=798156,-183832
EC00014=798156,-183832
EC00015=798156,-183832
EC00016=798156,-183832
EC00017=798156,-183832
EC00018=798156,-183832
EC00019=798156,-183832
EC00020=798156,-183832
EC00021=798156,-183832
EC00022=798156,-183832
EC00023=798156,-183832
EC00024=798156,-183832
EC00025=798156,-183832
EC00026=798156,-183832
EC00027=798156,-183832
EC00028=798156,-183832
EC00029=798156,-183832
EC00030=798156,-183832
EC00031=798156,-183832
EC00032=798156,-183832
EC00033=798156,-183832
EC00034=798156,-183832
EC00035=798156,-183832
EC00036=798156,-183832
EC00037=798156,-183832
EC00038=798156,-183832
EC00039=798156,-183832
EC00040=798156,-183832
EC00041=798156,-183832
EC00042=798156,-183832
EC00043=798156,-183832
EC00044=798156,-183832
EC00045=798156,-183832
EC00046=798156,-183832
EC00047=798156,-183832
EC00048=798156,-183832
EC00049=798156,-183832
EC00050=798156,-183832
EC00051=798156,-183832
EC00052=798156,-183832
EC00053=798156,-183832
EC00054=798156,-183832
EC00055=798156,-183832
EC00056=798156,-183832
EC00057=798156,-183832
EC00058=798156,-183832
EC00059=798156,-183832
EC00060=798156,-183832
EC00061=798156,-183832
EC00062=798156,-183832
EC00063=798156,-183832
EC00064=798156,-183832
EC00065=798156,-183832
EC00066=798156,-183832
EC00067=798156,-183832
EC00068=798156,-183832
EC00069=798156,-183832
EC00070=798156,-183832
EC00071=798156,-183832
EC00072=798156,-183832
EC00073=798156,-183832
EC00074=798156,-183832
EC00075=798156,-183832
EC00076=798156,-183832
EC00077=798156,-183832
EC00078=798156,-183832
EC00079=798156,-183832
EC00080=798156,-183832
EC00081=798156,-183832
EC00082=798156,-183832
EC00083=798156,-183832
EC00084=798156,-183832
EC00085=798156,-183832
EC00086=798156,-183832
EC00087=798156,-183832
EC00088=798156,-183832
EC00089=798156,-183832
EC00090=798156,-183832
EC00091=798156,-183832
EC00092=798156,-183832
EC00093=798156,-183832
EC00094=798156,-183832
EC00095=798156,-183832
EC00096=798156,-183832
EC00097=798156,-183832
EC00098=798156,-183832
EC00099=798156,-183832
EC00100=798156,-183832
EC00101=798156,-183832
EC00102=798156,-183832
EC00103=798156,-183832
EC00104=798156,-183832
EC00105=798156,-183832
EC00106=798156,-183832
EC00107=798156,-183832
EC00108=798156,-183832
EC00109=798156,-183832
EC00110=798156,-183832
EC00111=798156,-183832
EC00112=798156,-183832
EC00113=798156,-183832
EC00114=798156,-183832
EC00115=798156,-183832
EC00116=798156,-183832
EC00117=798156,-183832
EC00118=798156,-183832
EC00119=798156,-183832
EC00120=798156,-183832
EC00121=798156,-183832
EC00122=798156,-183832
EC00123=798156,-183832
EC00124=798156,-183832
EC00125=798156,-183832
EC00126=798156,-183832
EC00127=798156,-183832
EC00128=798155,-183832
EC00129=798152,-183831
EC00130=798155,-183832
EC00131=798155,-183832
EC00132=798155,-183832
EC00133=798156,-183832
EC00134=798156,-183832
EC00135=798156,-183832
EC00136=798156,-183832
EC00137=798156,-183832
EC00138=798156,-183832
EC00139=798156,-183832
EC00140=798156,-183832
EC00141=798156,-183832
EC00142=798156,-183832
EC00143=798156,-183832
EC00144=798156,-183832
EC00145=798156,-183832
EC00146=798156,-183832
EC00147=798156,-183832
EC00148=798156,-183832
EC00149=798156,-183832
EC00150=798156,-183832
EC00151=798156,-183832
EC00152=798156,-183832
EC00153=798156,-183832
EC00154=798156,-183832
EC00155=798156,-183832
EC00156=798156,-183832
EC00157=798156,-183832
EC00158=798156,-183832
EC00159=798156,-183832
EC00160=798156,-183832
EC00161=798156,-183832
EC00162=798156,-183832
EC00163=798156,-183832
EC00164=798156,-183832
EC00165=798156,-183832
EC00166=798156,-183832
EC00167=798156,-183832
EC00168=798156,-183832
EC00169=798156,-183832
EC00170=798156,-183832
EC00171=798156,-183832
EC00172=798156,-183832
EC00173=798156,-183832
EC00174=798156,-183832
EC00175=798156,-183832
EC00176=798156,-183832
EC00177=798156,-183832
EC00178=798156,-183832
EC00179=798156,-183832
EC00180=798156,-183832
EC00181=798156,-183832
EC00182=798156,-183832
EC00183=798156,-183832
EC00184=798156,-183832
EC00185=798156,-183832
EC00186=798156,-183832
EC00187=798156,-183832
EC00188=798156,-183832
EC00189=798156,-183832
EC00190=798156,-183832
EC00191=798156,-183832
EC00192=798156,-183832
EC00193=798156,-183832
EC00194=798156,-183832
EC00195=798156,-183832
EC00196=798156,-183832
EC00197=798156,-183832
EC00198=798156,-183832
EC00199=798156,-183832
EC00200=798156,-183832
EC00201=798156,-183832
EC00202=798156,-183832
EC00203=322978,-183832
EC00204=357094,925242
EC00205=800604,925242
EC00206=800604,925242
EC00207=800604,925242
EC00208=800603,925242
EC00209=800603,925242
EC00210=800603,925242
EC00211=800600,925239
EC00212=800600,925239
EC00213=800600,925239
EC00214=800600,925239
EC00215=800600,925239
EC00216=800600,925239
EC00217=800600,925239
EC00218=800600,925239
EC00219=800600,925239
EC00220=800600,925239
EC00221=800600,925239
EC00222=800600,925239
EC00223=800600,925239
EC00224=800600,925239
EC00225=800600,925239
EC00226=800600,925239
EC00227=800600,925239
EC00228=800600,925239
EC00229=800600,925239
EC00230=800600,925239
EC00231=800600,925239
EC00232=800600,925239
EC00233=800600,925239
EC00234=800600,925239
EC00235=800600,925239
EC00236=800600,925239
EC00237=800600,925239
EC00238=800600,925239
EC00239=800600,925239
EC00240=800600,925239
EC00241=800600,925239
EC00242=800600,925239
EC00243=800600,925239
EC00244=800600,925239
EC00245=800600,925239
EC00246=800600,925239
EC00247=800600,925239
EC00248=800600,925239
EC00249=800600,925239
EC00250=800600,925239
EC00251=800600,925239
EC00252=800600,925239
EC00253=800600,925239
EC00254=800600,925239
EC00255=800600,925239
EC00256=800600,925239
EC00257=800600,925239
EC00258=800600,925239
EC00259=800600,925239
EC00260=800600,925239
EC00261=800600,925239
EC00262=800600,925239
EC00263=800600,925239
EC00264=800600,925239
EC00265=800600,925239
EC00266=800600,925239
EC00267=800600,925239
EC00268=800600,925239
EC00269=800600,925239
EC00270=800600,925239
EC00271=800600,925239
EC00272=800600,925239
EC00273=800600,925239
EC00274=800600,925239
EC00275=800600,925239
EC00276=800600,925239
EC00277=800600,925239
EC00278=800600,925239
EC00279=800600,925239
EC00280=800600,925239
EC00281=800598,925237
EC00282=800598,925237
EC00283=800598,925237
EC00284=800598,925237
EC00285=800598,925237
EC00286=800598,925237
EC00287=800598,925237
EC00288=800598,925237
EC00289=800598,925237
EC00290=800598,925237
EC00291=800598,925237
EC00292=800598,925237
EC00293=800598,925237
EC00294=800598,925237
EC00295=800598,925237
EC00296=800598,925237
EC00297=800598,925237
EC00298=800598,925237
EC00299=800598,925237
EC00300=800598,925237
EC00301=800598,925237
EC00302=800598,925237
EC00303=800598,925237
EC00304=800598,925237
EC00305=800598,925237
EC00306=800600,925239
EC00307=800600,925239
EC00308=800600,925239
EC00309=800600,925239
EC00310=800600,925239
EC00311=800600,925239
EC00312=800600,925239
EC00313=800600,925239
EC00314=800603,925242
EC00315=800603,925242
EC00316=-11362,925242
EC00317=-11362,925242
EC00318=-798156,-183832
EC00319=-798156,-183832
EC00320=-798156,-183832
EC00321=-798156,-183832
EC00322=-798156,-183832
EC00323=-798156,-183832
EC00324=-798156,-183832
EC00325=-798156,-183832
EC00326=-798156,-183832
EC00327=-798156,-183832
EC00328=-798156,-183832
EC00329=-798156,-183832
EC00330=-798156,-183832
EC00331=-798156,-183832
EC00332=-798156,-183832
EC00333=-798156,-183832
EC00334=-798156,-183832
EC00335=-798156,-183832
EC00336=-798156,-183832
EC00337=-798156,-183832
EC00338=-798156,-183832
EC00339=-798156,-183832
EC00340=-798156,-183832
EC00341=-798156,-183832
EC00342=-798156,-183832
EC00343=-798156,-183832
EC00344=-798156,-183832
EC00345=-798156,-183832
EC00346=-798156,-183832
EC00347=-798156,-183832
EC00348=-798156,-183832
EC00349=-798156,-183832
EC00350=-798156,-183832
EC00351=-798156,-183832
EC00352=-798156,-183832
EC00353=-798156,-183832
EC00354=-798156,-183832
EC00355=-798156,-183832
EC00356=-798156,-183832
EC00357=-798156,-183832
EC00358=-798156,-183832
EC00359=-798156,-183832
EC00360=-798156,-183832
EC00361=-798156,-183832
EC00362=-798156,-183832
EC00363=-798156,-183832
EC00364=-798156,-183832
EC00365=-798156,-183832
EC00366=-798156,-183832
EC00367=-798156,-183832
EC00368=-798156,-183832
EC00369=-798156,-183832
EC00370=-798156,-183832
EC00371=-798156,-183832
EC00372=-798156,-183832
EC00373=-798156,-183832
EC00374=-798156,-183832
EC00375=-798156,-183832
EC00376=-798156,-183832
EC00377=-798156,-183832
EC00378=-798156,-183832
EC00379=-798156,-183832
EC00380=-798156,-183832
EC00381=-798156,-183832
EC00382=-798156,-183832
EC00383=-798156,-183832
EC00384=-798156,-183832
EC00385=-798156,-183832
EC00386=-798156,-183832
EC00387=-798156,-183832
EC00388=-798156,-183832
EC00389=-798156,-183832
EC00390=-798156,-183832
EC00391=-798156,-183832
EC00392=-798156,-183832
EC00393=-798156,-183832
EC00394=-798156,-183832
EC00395=-798156,-183832
EC00396=-798156,-183832
EC00397=-798156,-183832
EC00398=-798156,-183832
EC00399=-798156,-183832
EC00400=-798155,-183833
EC00401=-798155,-183833
EC00402=-798155,-183833
EC00403=-798156,-183832
EC00404=-798156,-183832
EC00405=-798156,-183832
EC00406=-798156,-183832
EC00407=-798156,-183832
EC00408=-798156,-183832
EC00409=-798156,-183832
EC00410=-798156,-183832
EC00411=-798156,-183832
EC00412=-798156,-183832
EC00413=-798156,-183832
EC00414=-798156,-183832
EC00415=-798156,-183832
EC00416=-798155,-183832
EC00417=-798156,-183832
EC00418=-798156,-183832
EC00419=-798156,-183832
EC00420=-798155,-183833
EC00421=-798156,-183832
EC00422=-798156,-183832
EC00423=-798156,-183832
EC00424=-798156,-183832
EC00425=-798156,-183832
EC00426=-798156,-183832
EC00427=-798156,-183832
EC00428=-798156,-183832
EC00429=-798156,-183832
EC00430=-798156,-183832
EC00431=-798156,-183832
EC00432=-798156,-183832
EC00433=-798156,-183832
EC00434=-798155,-183833
EC00435=-798156,-183832
EC00436=-798156,-183832
EC00437=-798156,-183832
EC00438=-798156,-183832
EC00439=-798156,-183832
EC00440=-798156,-183832
EC00441=-798156,-183832
EC00442=-798156,-183832
EC00443=-798156,-183832
EC00444=-798156,-183832
EC00445=-798156,-183832
EC00446=-798156,-183832
EC00447=-798156,-183832
EC00448=-798156,-183832
EC00449=-798156,-183832
EC00450=-798156,-183832
EC00451=-798156,-183832
EC00452=-798156,-183832
EC00453=-798156,-183832
EC00454=-798156,-183832
EC00455=-798156,-183832
EC00456=-798156,-183832
EC00457=-798156,-183832
EC00458=-798156,-183832
EC00459=-798156,-183832
EC00460=-798156,-183832
EC00461=-798156,-183832
EC00462=-798156,-183832
EC00463=-798156,-183832
EC00464=-798156,-183832
EC00465=-798156,-183832
EC00466=-798156,-183832
EC00467=-798156,-183832
EC00468=-798156,-183832
EC00469=-798156,-183832
EC00470=-798156,-183832
EC00471=-798156,-183832
EC00472=-798156,-183832
EC00473=-798156,-183832
EC00474=-798156,-183832
EC00475=-798156,-183832
EC00476=-798156,-183832
EC00477=-11362,925242
///POSTYPE BASE
///RECTAN
///RCONF 0,0,0,0,1,0,0,0,0,0,0,0,0,0,0,0,0,0,0,0,0,0,0,0
P00006=2.006,1.622,-0.565,0.0000,0.0000,0.0000
P00021=0.073,2.058,-0.109,0.0000,0.0000,0.0000
P00022=2.006,1.622,-0.565,0.0000,0.0000,0.0000
///RCONF 0,0,0,0,0,0,0,0,0,0,0,0,0,0,0,0,0,0,0,0,0,0,0,0
P00023=-2.957,-4.083,2.762,0.0000,0.0000,0.0000
P00024=-1.466,-0.226,-0.419,0.0000,0.0000,0.0000
P00025=3.643,0.007,-2.585,0.0000,0.0000,0.0000
P00026=2.644,0.055,-2.583,0.0000,0.0000,0.0000
P00027=2.278,0.099,-4.210,0.0000,0.0000,0.0000
P00028=-1.778,-0.182,-2.050,0.0000,0.0000,0.0000
P00029=1.749,4.006,-0.261,0.0000,0.0000,0.0000
P00031=-0.170,0.039,-0.647,0.0000,0.0000,0.0000
//INST
///DATE 2024/12/19 12:34
///ATTR SC,RW
///GROUP1 RB1,BS1
///GROUP2 ST1
NOP
'X2_34-37(-90,0)
'210,0
MOVJ C00000 BC00000 VJ=50.00  +MOVJ EC00000 VJ=50.00
MOVJ C00001 BC00001 VJ=100.00  +MOVJ EC00001 VJ=100.00
'Path S3633
SFTOF3D
MOVJ C00002 BC00002 VJ=50.00  +MOVJ EC00002 VJ=50.00
MOVJ C00003 BC00003 VJ=100.00  +MOVJ EC00003 VJ=100.00
MOVL C00004 BC00004 V=800.0  +MOVJ EC00004 VJ=100.00
SMOVL C00005 BC00005 V=166.7  +MOVJ EC00005
SREFP 3 C00006 BC00006  +REFP EC00006
CALL JOB:SEARCH-R1-S13D
SET P021 P006
SFTON3D P021
SMOVL C00007 BC00007 V=166.7  +MOVJ EC00007
SREFP 3 C00008 BC00008  +REFP EC00008
CALL JOB:SEARCH-R1-S13D
SET P021 P006
SFTON3D P021
SMOVL C00009 BC00009 V=166.7  +MOVJ EC00009
SMOVL C00010 BC00010 V=166.7  +MOVJ EC00010
SREFP 3 C00011 BC00011  +REFP EC00011
CALL JOB:SEARCH-R1-S13D
SET P021 P006
SFTON3D P021
SMOVL C00012 BC00012 V=166.7  +MOVJ EC00012
SFTOF3D
SMOVL C00013 BC00013 V=250.0  +MOVJ EC00013
SMOVL C00014 BC00014 V=166.7  +MOVJ EC00014
SREFP 3 C00015 BC00015  +REFP EC00015
CALL JOB:SEARCH-R1-S13D
SET P031 P006
SFTON3D P031
SMOVL C00016 BC00016 V=166.7  +MOVJ EC00016
SREFP 3 C00017 BC00017  +REFP EC00017
CALL JOB:SEARCH-R1-S13D
SET P031 P006
SFTON3D P031
SMOVL C00018 BC00018 V=166.7  +MOVJ EC00018
MOVL C00019 BC00019 V=800.0  +MOVJ EC00019 VJ=100.00
MOVL C00020 BC00020 V=1000.0  +MOVJ EC00020 VJ=100.00
'EndPath S3633
'Path S4258
SFTOF3D
MOVJ C00021 BC00021 VJ=100.00  +MOVJ EC00021 VJ=100.00
MOVL C00022 BC00022 V=800.0  +MOVJ EC00022 VJ=100.00
SMOVL C00023 BC00023 V=166.7  +MOVJ EC00023
SREFP 3 C00024 BC00024  +REFP EC00024
CALL JOB:SEARCH-R1-S13D
SET P022 P006
SFTON3D P022
SMOVL C00025 BC00025 V=166.7  +MOVJ EC00025
SMOVL C00026 BC00026 V=166.7  +MOVJ EC00026
SREFP 3 C00027 BC00027  +REFP EC00027
CALL JOB:SEARCH-R1-S13D
SET P022 P006
SFTON3D P022
SMOVL C00028 BC00028 V=166.7  +MOVJ EC00028
SMOVL C00029 BC00029 V=166.7  +MOVJ EC00029
SMOVL C00030 BC00030 V=166.7  +MOVJ EC00030
SREFP 3 C00031 BC00031  +REFP EC00031
CALL JOB:SEARCH-R1-S13D
SET P022 P006
SFTON3D P022
SMOVL C00032 BC00032 V=166.7  +MOVJ EC00032
SMOVL C00033 BC00033 V=166.7  +MOVJ EC00033
SMOVL C00034 BC00034 V=166.7  +MOVJ EC00034
MOVL C00035 BC00035 V=800.0  +MOVJ EC00035 VJ=100.00
MOVL C00036 BC00036 V=1000.0  +MOVJ EC00036 VJ=100.00
'EndPath S4258
'Path S4259
SFTOF3D
MOVJ C00037 BC00037 VJ=100.00  +MOVJ EC00037 VJ=100.00
MOVL C00038 BC00038 V=800.0  +MOVJ EC00038 VJ=100.00
SMOVL C00039 BC00039 V=166.7  +MOVJ EC00039
SREFP 3 C00040 BC00040  +REFP EC00040
CALL JOB:SEARCH-R1-S13D
SET P023 P006
SFTON3D P023
SMOVL C00041 BC00041 V=166.7  +MOVJ EC00041
SMOVL C00042 BC00042 V=166.7  +MOVJ EC00042
SREFP 3 C00043 BC00043  +REFP EC00043
CALL JOB:SEARCH-R1-S13D
SET P023 P006
SFTON3D P023
SMOVL C00044 BC00044 V=166.7  +MOVJ EC00044
SMOVL C00045 BC00045 V=166.7  +MOVJ EC00045
SREFP 3 C00046 BC00046  +REFP EC00046
CALL JOB:SEARCH-R1-S13D
SET P023 P006
SFTON3D P023
SMOVL C00047 BC00047 V=166.7  +MOVJ EC00047
MOVL C00048 BC00048 V=800.0  +MOVJ EC00048 VJ=100.00
MOVL C00049 BC00049 V=1000.0  +MOVJ EC00049 VJ=100.00
'EndPath S4259
'Path S4260
SFTOF3D
MOVJ C00050 BC00050 VJ=100.00  +MOVJ EC00050 VJ=100.00
MOVL C00051 BC00051 V=800.0  +MOVJ EC00051 VJ=100.00
SMOVL C00052 BC00052 V=166.7  +MOVJ EC00052
SREFP 3 C00053 BC00053  +REFP EC00053
CALL JOB:SEARCH-R1-S13D
SET P024 P006
SFTON3D P024
SMOVL C00054 BC00054 V=166.7  +MOVJ EC00054
SMOVL C00055 BC00055 V=166.7  +MOVJ EC00055
SREFP 3 C00056 BC00056  +REFP EC00056
CALL JOB:SEARCH-R1-S13D
SET P024 P006
SFTON3D P024
SMOVL C00057 BC00057 V=166.7  +MOVJ EC00057
SMOVL C00058 BC00058 V=166.7  +MOVJ EC00058
SMOVL C00059 BC00059 V=166.7  +MOVJ EC00059
SREFP 3 C00060 BC00060  +REFP EC00060
CALL JOB:SEARCH-R1-S13D
SET P024 P006
SFTON3D P024
SMOVL C00061 BC00061 V=166.7  +MOVJ EC00061
SMOVL C00062 BC00062 V=166.7  +MOVJ EC00062
SMOVL C00063 BC00063 V=166.7  +MOVJ EC00063
MOVL C00064 BC00064 V=800.0  +MOVJ EC00064 VJ=100.00
MOVL C00065 BC00065 V=1000.0  +MOVJ EC00065 VJ=100.00
'EndPath S4260
'Path S4261
SFTOF3D
MOVJ C00066 BC00066 VJ=100.00  +MOVJ EC00066 VJ=100.00
MOVL C00067 BC00067 V=800.0  +MOVJ EC00067 VJ=100.00
SMOVL C00068 BC00068 V=166.7  +MOVJ EC00068
SREFP 3 C00069 BC00069  +REFP EC00069
CALL JOB:SEARCH-R1-S13D
SET P025 P006
SFTON3D P025
SMOVL C00070 BC00070 V=166.7  +MOVJ EC00070
SMOVL C00071 BC00071 V=166.7  +MOVJ EC00071
SREFP 3 C00072 BC00072  +REFP EC00072
CALL JOB:SEARCH-R1-S13D
SET P025 P006
SFTON3D P025
SMOVL C00073 BC00073 V=166.7  +MOVJ EC00073
SMOVL C00074 BC00074 V=166.7  +MOVJ EC00074
SREFP 3 C00075 BC00075  +REFP EC00075
CALL JOB:SEARCH-R1-S13D
SET P025 P006
SFTON3D P025
SMOVL C00076 BC00076 V=166.7  +MOVJ EC00076
MOVL C00077 BC00077 V=800.0  +MOVJ EC00077 VJ=100.00
MOVL C00078 BC00078 V=1000.0  +MOVJ EC00078 VJ=100.00
'EndPath S4261
'Path S4262
SFTOF3D
MOVJ C00079 BC00079 VJ=100.00  +MOVJ EC00079 VJ=100.00
MOVL C00080 BC00080 V=800.0  +MOVJ EC00080 VJ=100.00
SMOVL C00081 BC00081 V=166.7  +MOVJ EC00081
SREFP 3 C00082 BC00082  +REFP EC00082
CALL JOB:SEARCH-R1-S13D
SET P026 P006
SFTON3D P026
SMOVL C00083 BC00083 V=166.7  +MOVJ EC00083
SMOVL C00084 BC00084 V=166.7  +MOVJ EC00084
SREFP 3 C00085 BC00085  +REFP EC00085
CALL JOB:SEARCH-R1-S13D
SET P026 P006
SFTON3D P026
SMOVL C00086 BC00086 V=166.7  +MOVJ EC00086
SMOVL C00087 BC00087 V=166.7  +MOVJ EC00087
SMOVL C00088 BC00088 V=166.7  +MOVJ EC00088
SREFP 3 C00089 BC00089  +REFP EC00089
CALL JOB:SEARCH-R1-S13D
SET P026 P006
SFTON3D P026
SMOVL C00090 BC00090 V=166.7  +MOVJ EC00090
SMOVL C00091 BC00091 V=166.7  +MOVJ EC00091
SMOVL C00092 BC00092 V=166.7  +MOVJ EC00092
MOVL C00093 BC00093 V=800.0  +MOVJ EC00093 VJ=100.00
MOVL C00094 BC00094 V=1000.0  +MOVJ EC00094 VJ=100.00
'EndPath S4262
'Path S4263
SFTOF3D
MOVJ C00095 BC00095 VJ=100.00  +MOVJ EC00095 VJ=100.00
MOVL C00096 BC00096 V=800.0  +MOVJ EC00096 VJ=100.00
SMOVL C00097 BC00097 V=166.7  +MOVJ EC00097
SREFP 3 C00098 BC00098  +REFP EC00098
CALL JOB:SEARCH-R1-S13D
SET P027 P006
SFTON3D P027
SMOVL C00099 BC00099 V=166.7  +MOVJ EC00099
SMOVL C00100 BC00100 V=166.7  +MOVJ EC00100
SREFP 3 C00101 BC00101  +REFP EC00101
CALL JOB:SEARCH-R1-S13D
SET P027 P006
SFTON3D P027
SMOVL C00102 BC00102 V=166.7  +MOVJ EC00102
SMOVL C00103 BC00103 V=166.7  +MOVJ EC00103
SMOVL C00104 BC00104 V=166.7  +MOVJ EC00104
SREFP 3 C00105 BC00105  +REFP EC00105
CALL JOB:SEARCH-R1-S13D
SET P027 P006
SFTON3D P027
SMOVL C00106 BC00106 V=166.7  +MOVJ EC00106
SMOVL C00107 BC00107 V=166.7  +MOVJ EC00107
SMOVL C00108 BC00108 V=166.7  +MOVJ EC00108
MOVL C00109 BC00109 V=800.0  +MOVJ EC00109 VJ=100.00
MOVL C00110 BC00110 V=1000.0  +MOVJ EC00110 VJ=100.00
'EndPath S4263
'
'Path W4264
SFTOF3D
SFTON3D P027
MOVJ C00111 BC00111 VJ=100.00  +MOVJ EC00111 VJ=100.00
MOVJ C00112 BC00112 VJ=100.00  +MOVJ EC00112 VJ=100.00
SMOVL C00113 BC00113 V=800.0  +MOVJ EC00113
SMOVL C00114 BC00114 V=150.0 PL=0  +MOVJ EC00114
MACRO1 MJ#(0) ARGF9
ARCON
SMOVL C00115 BC00115 V=10.0  +MOVJ EC00115
SMOVL C00116 BC00116 V=10.0  +MOVJ EC00116
SMOVL C00117 BC00117 V=7.5  +MOVJ EC00117
SMOVL C00118 BC00118 V=10.0  +MOVJ EC00118
ARCOF
SMOVL C00119 BC00119 V=800.0  +MOVJ EC00119
SMOVL C00120 BC00120 V=1000.0  +MOVJ EC00120
SFTOF3D
'EndPath W4264
MOVJ C00121 BC00121 VJ=100.00  +MOVJ EC00121 VJ=100.00
MOVJ C00122 BC00122 VJ=100.00  +MOVJ EC00122 VJ=100.00
MOVJ C00123 BC00123 VJ=100.00  +MOVJ EC00123 VJ=100.00
'Path W4265
SFTOF3D
SFTON3D P021
MOVJ C00124 BC00124 VJ=100.00  +MOVJ EC00124 VJ=100.00
SMOVL C00125 BC00125 V=800.0  +MOVJ EC00125
SMOVL C00126 BC00126 V=150.0 PL=0  +MOVJ EC00126
ARCON
SMOVL C00127 BC00127 V=10.0  +MOVJ EC00127
SMOVL C00128 BC00128 V=7.5  +MOVJ EC00128
SMOVL C00129 BC00129 V=7.5  +MOVJ EC00129
SFTON3D P031
SMOVL C00130 BC00130 V=9.2  +MOVJ EC00130
SMOVL C00131 BC00131 V=9.2  +MOVJ EC00131
ARCOF
SMOVL C00132 BC00132 V=250.0  +MOVJ EC00132
SMOVL C00133 BC00133 V=800.0  +MOVJ EC00133
SMOVL C00134 BC00134 V=1000.0  +MOVJ EC00134
SFTOF3D
'EndPath W4265
MOVJ C00135 BC00135 VJ=100.00  +MOVJ EC00135 VJ=100.00
MOVJ C00136 BC00136 VJ=100.00  +MOVJ EC00136 VJ=100.00
MOVJ C00137 BC00137 VJ=100.00  +MOVJ EC00137 VJ=100.00
'Path W4266
SFTOF3D
SFTON3D P025
MOVJ C00138 BC00138 VJ=100.00  +MOVJ EC00138 VJ=100.00
SMOVL C00139 BC00139 V=800.0  +MOVJ EC00139
SMOVL C00140 BC00140 V=150.0 PL=0  +MOVJ EC00140
ARCON
SMOVL C00141 BC00141 V=9.2  +MOVJ EC00141
SMOVL C00142 BC00142 V=9.2  +MOVJ EC00142
SMOVL C00143 BC00143 V=10.0  +MOVJ EC00143
SMOVL C00144 BC00144 V=9.2  +MOVJ EC00144
SMOVL C00145 BC00145 V=9.2  +MOVJ EC00145
SMOVL C00146 BC00146 V=9.2  +MOVJ EC00146
ARCOF
SMOVL C00147 BC00147 V=800.0  +MOVJ EC00147
SMOVL C00148 BC00148 V=1000.0  +MOVJ EC00148
SFTOF3D
'EndPath W4266
MOVJ C00149 BC00149 VJ=100.00  +MOVJ EC00149 VJ=100.00
MOVJ C00150 BC00150 VJ=100.00  +MOVJ EC00150 VJ=100.00
MOVJ C00151 BC00151 VJ=100.00  +MOVJ EC00151 VJ=100.00
'Path W4267
SFTOF3D
SFTON3D P023
MOVJ C00152 BC00152 VJ=100.00  +MOVJ EC00152 VJ=100.00
SMOVL C00153 BC00153 V=800.0  +MOVJ EC00153
SMOVL C00154 BC00154 V=150.0 PL=0  +MOVJ EC00154
ARCON
SMOVL C00155 BC00155 V=9.2  +MOVJ EC00155
SMOVL C00156 BC00156 V=9.2  +MOVJ EC00156
SMOVL C00157 BC00157 V=9.2  +MOVJ EC00157
SMOVL C00158 BC00158 V=9.2  +MOVJ EC00158
SMOVL C00159 BC00159 V=9.2  +MOVJ EC00159
SMOVL C00160 BC00160 V=9.2  +MOVJ EC00160
ARCOF
SMOVL C00161 BC00161 V=800.0  +MOVJ EC00161
SMOVL C00162 BC00162 V=1000.0  +MOVJ EC00162
SFTOF3D
'EndPath W4267
MOVJ C00163 BC00163 VJ=100.00  +MOVJ EC00163 VJ=100.00
MOVJ C00164 BC00164 VJ=100.00  +MOVJ EC00164 VJ=100.00
'
'Path W4268
SFTOF3D
SFTON3D P026
MOVJ C00165 BC00165 VJ=100.00  +MOVJ EC00165 VJ=100.00
SMOVL C00166 BC00166 V=800.0  +MOVJ EC00166
SMOVL C00167 BC00167 V=150.0 PL=0  +MOVJ EC00167
ARCON
SMOVL C00168 BC00168 V=9.2  +MOVJ EC00168
SMOVL C00169 BC00169 V=9.2  +MOVJ EC00169
SMOVL C00170 BC00170 V=9.2  +MOVJ EC00170
SMOVL C00171 BC00171 V=9.2  +MOVJ EC00171
ARCOF
SMOVL C00172 BC00172 V=800.0  +MOVJ EC00172
SMOVL C00173 BC00173 V=1000.0  +MOVJ EC00173
SFTOF3D
'EndPath W4268
MOVJ C00174 BC00174 VJ=100.00  +MOVJ EC00174 VJ=100.00
MOVJ C00175 BC00175 VJ=100.00  +MOVJ EC00175 VJ=100.00
MOVJ C00176 BC00176 VJ=100.00  +MOVJ EC00176 VJ=100.00
'Path W3636
SFTOF3D
SFTON3D P022
MOVJ C00177 BC00177 VJ=100.00  +MOVJ EC00177 VJ=100.00
SMOVL C00178 BC00178 V=800.0  +MOVJ EC00178
SMOVL C00179 BC00179 V=150.0 PL=0  +MOVJ EC00179
ARCON
SMOVL C00180 BC00180 V=9.2  +MOVJ EC00180
SMOVL C00181 BC00181 V=9.2  +MOVJ EC00181
SMOVL C00182 BC00182 V=9.2  +MOVJ EC00182
SMOVL C00183 BC00183 V=9.2  +MOVJ EC00183
SMOVL C00184 BC00184 V=9.2  +MOVJ EC00184
SMOVL C00185 BC00185 V=9.2  +MOVJ EC00185
ARCOF
SMOVL C00186 BC00186 V=800.0  +MOVJ EC00186
SMOVL C00187 BC00187 V=1000.0  +MOVJ EC00187
SFTOF3D
'EndPath W3636
'Path W4269
SFTOF3D
SFTON3D P024
MOVJ C00188 BC00188 VJ=100.00  +MOVJ EC00188 VJ=100.00
SMOVL C00189 BC00189 V=800.0  +MOVJ EC00189
SMOVL C00190 BC00190 V=150.0 PL=0  +MOVJ EC00190
ARCON
SMOVL C00191 BC00191 V=9.2  +MOVJ EC00191
SMOVL C00192 BC00192 V=9.2  +MOVJ EC00192
SMOVL C00193 BC00193 V=9.2  +MOVJ EC00193
SMOVL C00194 BC00194 V=9.2  +MOVJ EC00194
SMOVL C00195 BC00195 V=9.2  +MOVJ EC00195
SMOVL C00196 BC00196 V=9.2  +MOVJ EC00196
ARCOF
SMOVL C00197 BC00197 V=800.0  +MOVJ EC00197
SMOVL C00198 BC00198 V=1000.0  +MOVJ EC00198
SFTOF3D
'EndPath W4269
MOVJ C00199 BC00199 VJ=100.00  +MOVJ EC00199 VJ=100.00
MOVJ C00200 BC00200 VJ=100.00  +MOVJ EC00200 VJ=100.00
MOVJ C00201 BC00201 VJ=100.00  +MOVJ EC00201 VJ=100.00
CALL JOB:CLEAN-R1_KM_NEW
'
'
'
'Cut-Wire
MOVJ C00202 BC00202 VJ=100.00  +MOVJ EC00202 VJ=100.00
MOVJ C00203 BC00203 VJ=100.00  +MOVJ EC00203 VJ=100.00
MOVJ C00204 BC00204 VJ=100.00  +MOVJ EC00204 VJ=100.00
MOVJ C00205 BC00205 VJ=100.00  +MOVJ EC00205 VJ=100.00
MOVJ C00206 BC00206 VJ=100.00  +MOVJ EC00206 VJ=100.00
MOVJ C00207 BC00207 VJ=100.00  +MOVJ EC00207 VJ=100.00
MOVJ C00208 BC00208 VJ=30.00  +MOVJ EC00208 VJ=100.00
MOVL C00209 BC00209 V=333.3  +MOVJ EC00209 VJ=30.00
MOVL C00210 BC00210 V=333.3  +MOVJ EC00210 VJ=30.00
SFTOF3D
SMOVL C00211 BC00211 V=166.7  +MOVJ EC00211
SREFP 3 C00212 BC00212  +REFP EC00212
CALL JOB:SEARCH-R1-S13D
SET P027 P006
SFTON3D P027
SMOVL C00213 BC00213 V=166.7  +MOVJ EC00213
SREFP 3 C00214 BC00214  +REFP EC00214
CALL JOB:SEARCH-R1-S13D
SET P027 P006
SFTON3D P027
SMOVL C00215 BC00215 V=166.7  +MOVJ EC00215
SFTOF3D
MOVL C00216 BC00216 V=333.3  +MOVJ EC00216 VJ=30.00
SFTOF3D
SMOVL C00217 BC00217 V=166.7  +MOVJ EC00217
SREFP 3 C00218 BC00218  +REFP EC00218
CALL JOB:SEARCH-R1-S13D
SET P026 P006
SFTON3D P026
SMOVL C00219 BC00219 V=166.7  +MOVJ EC00219
SREFP 3 C00220 BC00220  +REFP EC00220
CALL JOB:SEARCH-R1-S13D
SET P026 P006
SFTON3D P026
SMOVL C00221 BC00221 V=166.7  +MOVJ EC00221
SFTOF3D
SMOVL C00222 BC00222 V=166.7  +MOVJ EC00222
SREFP 3 C00223 BC00223  +REFP EC00223
CALL JOB:SEARCH-R1-S13D
SET P025 P006
SFTON3D P025
SMOVL C00224 BC00224 V=166.7  +MOVJ EC00224
SREFP 3 C00225 BC00225  +REFP EC00225
CALL JOB:SEARCH-R1-S13D
SET P025 P006
SFTON3D P025
SMOVL C00226 BC00226 V=166.7  +MOVJ EC00226
SFTOF3D
SMOVL C00227 BC00227 V=166.7  +MOVJ EC00227
SREFP 3 C00228 BC00228  +REFP EC00228
CALL JOB:SEARCH-R1-S13D
SET P024 P006
SFTON3D P024
SMOVL C00229 BC00229 V=166.7  +MOVJ EC00229
SREFP 3 C00230 BC00230  +REFP EC00230
CALL JOB:SEARCH-R1-S13D
SET P024 P006
SFTON3D P024
SMOVL C00231 BC00231 V=166.7  +MOVJ EC00231
SFTOF3D
MOVL C00232 BC00232 V=333.3  +MOVJ EC00232 VJ=30.00
SMOVL C00233 BC00233 V=166.7  +MOVJ EC00233
SREFP 3 C00234 BC00234  +REFP EC00234
CALL JOB:SEARCH-R1-S13D
SET P028 P006
SFTON3D P028
SMOVL C00235 BC00235 V=166.7  +MOVJ EC00235
SREFP 3 C00236 BC00236  +REFP EC00236
CALL JOB:SEARCH-R1-S13D
SET P028 P006
SFTON3D P028
SMOVL C00237 BC00237 V=166.7  +MOVJ EC00237
SFTOF3D
SMOVL C00238 BC00238 V=166.7  +MOVJ EC00238
SREFP 3 C00239 BC00239  +REFP EC00239
CALL JOB:SEARCH-R1-S13D
SET P023 P006
SFTON3D P023
SMOVL C00240 BC00240 V=166.7  +MOVJ EC00240
SREFP 3 C00241 BC00241  +REFP EC00241
CALL JOB:SEARCH-R1-S13D
SET P023 P006
SFTON3D P023
SMOVL C00242 BC00242 V=166.7  +MOVJ EC00242
SFTOF3D
MOVJ C00243 BC00243 VJ=50.00  +MOVJ EC00243 VJ=50.00
MOVJ C00244 BC00244 VJ=30.00  +MOVJ EC00244 VJ=30.00
SMOVL C00245 BC00245 V=166.7  +MOVJ EC00245
SREFP 3 C00246 BC00246  +REFP EC00246
CALL JOB:SEARCH-R1-S13D
SET P029 P006
SFTON3D P029
SMOVL C00247 BC00247 V=166.7  +MOVJ EC00247
SREFP 3 C00248 BC00248  +REFP EC00248
CALL JOB:SEARCH-R1-S13D
SET P029 P006
SFTON3D P029
SMOVL C00249 BC00249 V=166.7  +MOVJ EC00249
SFTOF3D
MOVL C00250 BC00250 V=333.3  +MOVJ EC00250 VJ=30.00
MOVL C00251 BC00251 V=333.3  +MOVJ EC00251 VJ=30.00
SMOVL C00252 BC00252 V=166.7  +MOVJ EC00252
SREFP 3 C00253 BC00253  +REFP EC00253
CALL JOB:SEARCH-R1-S13D
SET P022 P006
SFTON3D P022
SMOVL C00254 BC00254 V=166.7  +MOVJ EC00254
SREFP 3 C00255 BC00255  +REFP EC00255
CALL JOB:SEARCH-R1-S13D
SET P022 P006
SFTON3D P022
SMOVL C00256 BC00256 V=166.7  +MOVJ EC00256
SFTOF3D
MOVL C00257 BC00257 V=333.3  +MOVJ EC00257 VJ=30.00
SMOVL C00258 BC00258 V=166.7  +MOVJ EC00258
SREFP 3 C00259 BC00259  +REFP EC00259
CALL JOB:SEARCH-R1-S13D
SET P021 P006
SFTON3D P021
SMOVL C00260 BC00260 V=166.7  +MOVJ EC00260
SREFP 3 C00261 BC00261  +REFP EC00261
CALL JOB:SEARCH-R1-S13D
SET P021 P006
SFTON3D P021
SMOVL C00262 BC00262 V=166.7  +MOVJ EC00262
SMOVL C00263 BC00263 V=166.7  +MOVJ EC00263
MACRO1 MJ#(0) ARGF9
SFTON3D P022
SMOVL C00264 BC00264 V=166.7  +MOVJ EC00264
ARCON
SMOVL C00265 BC00265 V=10.0  +MOVJ EC00265
SMOVL C00266 BC00266 V=10.0  +MOVJ EC00266
SFTON3D P021
SMOVL C00267 BC00267 V=10.0  +MOVJ EC00267
SMOVL C00268 BC00268 V=10.0  +MOVJ EC00268
SMOVL C00269 BC00269 V=10.0  +MOVJ EC00269
SMOVL C00270 BC00270 V=10.0  +MOVJ EC00270
ARCOF
SFTOF3D
SMOVL C00271 BC00271 V=250.0  +MOVJ EC00271
SMOVL C00272 BC00272 V=250.0  +MOVJ EC00272
MOVJ C00273 BC00273 VJ=30.00  +MOVJ EC00273 VJ=30.00
SMOVL C00274 BC00274 V=250.0  +MOVJ EC00274
SFTON3D P029
SMOVL C00275 BC00275 V=250.0  +MOVJ EC00275
ARCON
SMOVL C00276 BC00276 V=10.0  +MOVJ EC00276
SMOVL C00277 BC00277 V=10.0  +MOVJ EC00277
SMOVL C00278 BC00278 V=10.0  +MOVJ EC00278
SMOVL C00279 BC00279 V=10.0  +MOVJ EC00279
ARCOF
SFTOF3D
SMOVL C00280 BC00280 V=333.3  +MOVJ EC00280
SMOVL C00281 BC00281 V=333.3  +MOVJ EC00281
SFTON3D P028
SMOVL C00282 BC00282 V=250.0  +MOVJ EC00282
ARCON
SMOVL C00283 BC00283 V=10.0  +MOVJ EC00283
SMOVL C00284 BC00284 V=10.0  +MOVJ EC00284
SMOVL C00285 BC00285 V=10.0  +MOVJ EC00285
SFTON3D P023
SMOVL C00286 BC00286 V=10.0  +MOVJ EC00286
SMOVL C00287 BC00287 V=10.0  +MOVJ EC00287
ARCOF
SFTOF3D
SMOVL C00288 BC00288 V=333.3  +MOVJ EC00288
SMOVL C00289 BC00289 V=333.3  +MOVJ EC00289
SFTON3D P024
SMOVL C00290 BC00290 V=166.7  +MOVJ EC00290
ARCON
SMOVL C00291 BC00291 V=10.0  +MOVJ EC00291
SMOVL C00292 BC00292 V=10.0  +MOVJ EC00292
SMOVL C00293 BC00293 V=10.0  +MOVJ EC00293
SMOVL C00294 BC00294 V=10.0  +MOVJ EC00294
SMOVL C00295 BC00295 V=10.0  +MOVJ EC00295
ARCOF
SFTOF3D
SMOVL C00296 BC00296 V=250.0  +MOVJ EC00296
SMOVL C00297 BC00297 V=250.0  +MOVJ EC00297
SFTON3D P026
SMOVL C00298 BC00298 V=250.0  +MOVJ EC00298
ARCON
SMOVL C00299 BC00299 V=10.0  +MOVJ EC00299
SMOVL C00300 BC00300 V=10.0  +MOVJ EC00300
SFTON3D P025
SMOVL C00301 BC00301 V=10.0  +MOVJ EC00301
SMOVL C00302 BC00302 V=10.0  +MOVJ EC00302
SMOVL C00303 BC00303 V=10.0  +MOVJ EC00303
ARCOF
SFTOF3D
SMOVL C00304 BC00304 V=250.0  +MOVJ EC00304
'do sprawdzenia
PAUSE
SMOVL C00305 BC00305 V=250.0  +MOVJ EC00305
SFTON3D P027
SMOVL C00306 BC00306 V=250.0  +MOVJ EC00306
ARCON
SMOVL C00307 BC00307 V=10.0  +MOVJ EC00307
SMOVL C00308 BC00308 V=10.0  +MOVJ EC00308
SMOVL C00309 BC00309 V=10.0  +MOVJ EC00309
SMOVL C00310 BC00310 V=10.0  +MOVJ EC00310
SMOVL C00311 BC00311 V=10.0  +MOVJ EC00311
SMOVL C00312 BC00312 V=10.0  +MOVJ EC00312
ARCOF
SFTOF3D
SMOVL C00313 BC00313 V=250.0  +MOVJ EC00313
SMOVL C00314 BC00314 V=250.0  +MOVJ EC00314
MOVJ C00315 BC00315 VJ=30.00  +MOVJ EC00315 VJ=30.00
MOVJ C00316 BC00316 VJ=100.00  +MOVJ EC00316 VJ=100.00
MOVJ C00317 BC00317 VJ=100.00  +MOVJ EC00317 VJ=100.00
COMM MOVJ C00318 BC00318 VJ=100.00  +MOVJ EC00318 VJ=100.00
COMM MOVJ C00319 BC00319 VJ=100.00  +MOVJ EC00319 VJ=100.00
'obrot
COMM MOVJ C00320 BC00320 VJ=100.00  +MOVJ EC00320 VJ=100.00
COMM MOVJ C00321 BC00321 VJ=100.00  +MOVJ EC00321 VJ=100.00
COMM MOVJ C00322 BC00322 VJ=100.00  +MOVJ EC00322 VJ=100.00
COMM 'Path S4271
COMM SFTOF3D
COMM MOVJ C00323 BC00323 VJ=100.00  +MOVJ EC00323 VJ=100.00
COMM MOVL C00324 BC00324 V=800.0  +MOVJ EC00324 VJ=100.00
COMM SMOVL C00325 BC00325 V=166.7  +MOVJ EC00325
COMM SREFP 3 C00326 BC00326  +REFP EC00326
COMM CALL JOB:SEARCH-R1-S13D
COMM SET P021 P006
COMM SFTON3D P021
COMM SMOVL C00327 BC00327 V=166.7  +MOVJ EC00327
COMM SREFP 3 C00328 BC00328  +REFP EC00328
COMM CALL JOB:SEARCH-R1-S13D
COMM SET P021 P006
COMM SFTON3D P021
COMM SMOVL C00329 BC00329 V=166.7  +MOVJ EC00329
COMM 'EndPath S4271
COMM 'Path S4272
COMM SFTOF3D
COMM MOVJ C00330 BC00330 VJ=100.00  +MOVJ EC00330 VJ=100.00
COMM SMOVL C00331 BC00331 V=166.7  +MOVJ EC00331
COMM SREFP 3 C00332 BC00332  +REFP EC00332
COMM CALL JOB:SEARCH-R1-S13D
COMM SET P022 P006
COMM SFTON3D P022
COMM SMOVL C00333 BC00333 V=166.7  +MOVJ EC00333
COMM SMOVL C00334 BC00334 V=166.7  +MOVJ EC00334
COMM SREFP 3 C00335 BC00335  +REFP EC00335
COMM CALL JOB:SEARCH-R1-S13D
COMM SET P022 P006
COMM SFTON3D P022
COMM SMOVL C00336 BC00336 V=166.7  +MOVJ EC00336
COMM SMOVL C00337 BC00337 V=166.7  +MOVJ EC00337
COMM SMOVL C00338 BC00338 V=166.7  +MOVJ EC00338
COMM SREFP 3 C00339 BC00339  +REFP EC00339
COMM CALL JOB:SEARCH-R1-S13D
COMM SET P022 P006
COMM SFTON3D P022
COMM SMOVL C00340 BC00340 V=166.7  +MOVJ EC00340
COMM 'EndPath S4272
COMM 'Path S4273
COMM SFTOF3D
COMM MOVL C00341 BC00341 V=800.0  +MOVJ EC00341 VJ=100.00
COMM SMOVL C00342 BC00342 V=166.7  +MOVJ EC00342
COMM SREFP 3 C00343 BC00343  +REFP EC00343
COMM CALL JOB:SEARCH-R1-S13D
COMM SET P023 P006
COMM SFTON3D P023
COMM SMOVL C00344 BC00344 V=166.7  +MOVJ EC00344
COMM SREFP 3 C00345 BC00345  +REFP EC00345
COMM CALL JOB:SEARCH-R1-S13D
COMM SET P023 P006
COMM SFTON3D P023
COMM SMOVL C00346 BC00346 V=166.7  +MOVJ EC00346
COMM SMOVL C00347 BC00347 V=166.7  +MOVJ EC00347
COMM SREFP 3 C00348 BC00348  +REFP EC00348
COMM CALL JOB:SEARCH-R1-S13D
COMM SET P023 P006
COMM SFTON3D P023
COMM SMOVL C00349 BC00349 V=166.7  +MOVJ EC00349
COMM MOVL C00350 BC00350 V=1000.0  +MOVJ EC00350 VJ=100.00
COMM 'EndPath S4273
COMM 'Path S4274
COMM SFTOF3D
COMM MOVJ C00351 BC00351 VJ=100.00  +MOVJ EC00351 VJ=100.00
COMM SMOVL C00352 BC00352 V=166.7  +MOVJ EC00352
COMM SREFP 3 C00353 BC00353  +REFP EC00353
COMM CALL JOB:SEARCH-R1-S13D
COMM SET P024 P006
COMM SFTON3D P024
COMM SMOVL C00354 BC00354 V=166.7  +MOVJ EC00354
COMM SREFP 3 C00355 BC00355  +REFP EC00355
COMM CALL JOB:SEARCH-R1-S13D
COMM SET P024 P006
COMM SFTON3D P024
COMM SMOVL C00356 BC00356 V=166.7  +MOVJ EC00356
COMM SMOVL C00357 BC00357 V=166.7  +MOVJ EC00357
COMM SMOVL C00358 BC00358 V=166.7  +MOVJ EC00358
COMM SREFP 3 C00359 BC00359  +REFP EC00359
COMM CALL JOB:SEARCH-R1-S13D
COMM SET P024 P006
COMM SFTON3D P024
COMM SMOVL C00360 BC00360 V=166.7  +MOVJ EC00360
COMM 'EndPath S4274
COMM 'Path S4275
COMM SFTOF3D
COMM MOVL C00361 BC00361 V=800.0  +MOVJ EC00361 VJ=100.00
COMM SMOVL C00362 BC00362 V=166.7  +MOVJ EC00362
COMM SREFP 3 C00363 BC00363  +REFP EC00363
COMM CALL JOB:SEARCH-R1-S13D
COMM SET P025 P006
COMM SFTON3D P025
COMM SMOVL C00364 BC00364 V=166.7  +MOVJ EC00364
COMM SMOVL C00365 BC00365 V=166.7  +MOVJ EC00365
COMM SREFP 3 C00366 BC00366  +REFP EC00366
COMM CALL JOB:SEARCH-R1-S13D
COMM SET P025 P006
COMM SFTON3D P025
COMM SMOVL C00367 BC00367 V=166.7  +MOVJ EC00367
COMM SMOVL C00368 BC00368 V=166.7  +MOVJ EC00368
COMM SREFP 3 C00369 BC00369  +REFP EC00369
COMM CALL JOB:SEARCH-R1-S13D
COMM SET P025 P006
COMM SFTON3D P025
COMM SMOVL C00370 BC00370 V=166.7  +MOVJ EC00370
COMM SFTOF3D
COMM SMOVL C00371 BC00371 V=250.0  +MOVJ EC00371
COMM SREFP 3 C00372 BC00372  +REFP EC00372
COMM CALL JOB:SEARCH-R1-S13D
COMM SET P026 P006
COMM SFTON3D P026
COMM SMOVL C00373 BC00373 V=166.7  +MOVJ EC00373
COMM SREFP 3 C00374 BC00374  +REFP EC00374
COMM CALL JOB:SEARCH-R1-S13D
COMM SET P026 P006
COMM SFTON3D P026
COMM SMOVL C00375 BC00375 V=166.7  +MOVJ EC00375
COMM SMOVL C00376 BC00376 V=250.0  +MOVJ EC00376
COMM SMOVL C00377 BC00377 V=166.7  +MOVJ EC00377
COMM SREFP 3 C00378 BC00378  +REFP EC00378
COMM CALL JOB:SEARCH-R1-S13D
COMM SET P026 P006
COMM SFTON3D P026
COMM SMOVL C00379 BC00379 V=166.7  +MOVJ EC00379
COMM 'EndPath S4276
COMM 'Path S4277
COMM SFTOF3D
COMM MOVL C00380 BC00380 V=800.0  +MOVJ EC00380 VJ=100.00
COMM SMOVL C00381 BC00381 V=166.7  +MOVJ EC00381
COMM SREFP 3 C00382 BC00382  +REFP EC00382
COMM CALL JOB:SEARCH-R1-S13D
COMM SET P027 P006
COMM SFTON3D P027
COMM SMOVL C00383 BC00383 V=166.7  +MOVJ EC00383
COMM SMOVL C00384 BC00384 V=166.7  +MOVJ EC00384
COMM SREFP 3 C00385 BC00385  +REFP EC00385
COMM CALL JOB:SEARCH-R1-S13D
COMM SET P027 P006
COMM SFTON3D P027
COMM SMOVL C00386 BC00386 V=166.7  +MOVJ EC00386
COMM SMOVL C00387 BC00387 V=166.7  +MOVJ EC00387
COMM SMOVL C00388 BC00388 V=166.7  +MOVJ EC00388
COMM SREFP 3 C00389 BC00389  +REFP EC00389
COMM CALL JOB:SEARCH-R1-S13D
COMM SET P027 P006
COMM SFTON3D P027
COMM SMOVL C00390 BC00390 V=166.7  +MOVJ EC00390
COMM SMOVL C00391 BC00391 V=166.7  +MOVJ EC00391
COMM SMOVL C00392 BC00392 V=166.7  +MOVJ EC00392
COMM MOVL C00393 BC00393 V=800.0  +MOVJ EC00393 VJ=100.00
COMM MOVL C00394 BC00394 V=500.0  +MOVJ EC00394 VJ=100.00
COMM 'EndPath S4277
COMM '
COMM 'Path W4278
COMM SFTOF3D
COMM SFTON3D P027
COMM MOVJ C00395 BC00395 VJ=40.00  +MOVJ EC00395 VJ=100.00
COMM SMOVL C00396 BC00396 V=800.0  +MOVJ EC00396
COMM SMOVL C00397 BC00397 V=150.0 PL=0  +MOVJ EC00397
COMM ARCON
COMM SMOVL C00398 BC00398 V=10.0  +MOVJ EC00398
COMM SMOVL C00399 BC00399 V=10.0  +MOVJ EC00399
COMM ARCOF
COMM SMOVL C00400 BC00400 V=800.0  +MOVJ EC00400
COMM SMOVL C00401 BC00401 V=1000.0  +MOVJ EC00401
COMM SFTOF3D
COMM 'EndPath W4278
COMM MOVJ C00402 BC00402 VJ=100.00  +MOVJ EC00402 VJ=100.00
COMM MOVJ C00403 BC00403 VJ=100.00  +MOVJ EC00403 VJ=100.00
COMM MOVJ C00404 BC00404 VJ=100.00  +MOVJ EC00404 VJ=100.00
COMM 'Path W4279
COMM SFTOF3D
COMM SFTON3D P021
COMM MOVJ C00405 BC00405 VJ=100.00  +MOVJ EC00405 VJ=100.00
COMM SMOVL C00406 BC00406 V=800.0  +MOVJ EC00406
COMM SMOVL C00407 BC00407 V=150.0 PL=0  +MOVJ EC00407
COMM SMOVL C00408 BC00408 V=10.0  +MOVJ EC00408
COMM SMOVL C00409 BC00409 V=10.0  +MOVJ EC00409
COMM SMOVL C00410 BC00410 V=10.0  +MOVJ EC00410
COMM ARCOF
COMM SMOVL C00411 BC00411 V=800.0  +MOVJ EC00411
COMM SMOVL C00412 BC00412 V=1000.0  +MOVJ EC00412
COMM SFTOF3D
COMM 'EndPath W4279
COMM MOVJ C00413 BC00413 VJ=100.00  +MOVJ EC00413 VJ=100.00
COMM SMOVL C00414 BC00414 V=500.0  +MOVJ EC00414
COMM 'Path W4280
COMM SFTOF3D
COMM SFTON3D P025
COMM SMOVL C00415 BC00415 V=800.0  +MOVJ EC00415
COMM SMOVL C00416 BC00416 V=150.0 PL=0  +MOVJ EC00416
COMM ARCON
COMM SMOVL C00417 BC00417 V=10.0  +MOVJ EC00417
COMM SMOVL C00418 BC00418 V=10.0  +MOVJ EC00418
COMM SMOVL C00419 BC00419 V=10.0  +MOVJ EC00419
COMM SMOVL C00420 BC00420 V=10.0  +MOVJ EC00420
COMM SMOVL C00421 BC00421 V=10.0  +MOVJ EC00421
COMM SMOVL C00422 BC00422 V=10.0  +MOVJ EC00422
COMM ARCOF
COMM SMOVL C00423 BC00423 V=800.0  +MOVJ EC00423
COMM SMOVL C00424 BC00424 V=1000.0  +MOVJ EC00424
COMM SFTOF3D
COMM 'EndPath W4280
COMM MOVJ C00425 BC00425 VJ=100.00  +MOVJ EC00425 VJ=100.00
COMM 'Path W4281
COMM SFTOF3D
COMM SFTON3D P023
COMM MOVJ C00426 BC00426 VJ=100.00  +MOVJ EC00426 VJ=100.00
COMM SMOVL C00427 BC00427 V=800.0  +MOVJ EC00427
COMM SMOVL C00428 BC00428 V=150.0 PL=0  +MOVJ EC00428
COMM ARCON
COMM SMOVL C00429 BC00429 V=10.0  +MOVJ EC00429
COMM SMOVL C00430 BC00430 V=10.0  +MOVJ EC00430
COMM SMOVL C00431 BC00431 V=10.0  +MOVJ EC00431
COMM SMOVL C00432 BC00432 V=10.0  +MOVJ EC00432
COMM SMOVL C00433 BC00433 V=10.0  +MOVJ EC00433
COMM SMOVL C00434 BC00434 V=10.0  +MOVJ EC00434
COMM ARCOF
COMM SMOVL C00435 BC00435 V=800.0  +MOVJ EC00435
COMM SMOVL C00436 BC00436 V=1000.0  +MOVJ EC00436
COMM SFTOF3D
COMM 'EndPath W4281
COMM MOVJ C00437 BC00437 VJ=100.00  +MOVJ EC00437 VJ=100.00
COMM '
COMM 'Path W4282
COMM SFTOF3D
COMM SFTON3D P026
COMM MOVJ C00438 BC00438 VJ=100.00  +MOVJ EC00438 VJ=100.00
COMM SMOVL C00439 BC00439 V=800.0  +MOVJ EC00439
COMM SMOVL C00440 BC00440 V=150.0 PL=0  +MOVJ EC00440
COMM ARCON
COMM SMOVL C00441 BC00441 V=10.0  +MOVJ EC00441
COMM SMOVL C00442 BC00442 V=10.0  +MOVJ EC00442
COMM SMOVL C00443 BC00443 V=10.0  +MOVJ EC00443
COMM SMOVL C00444 BC00444 V=10.0  +MOVJ EC00444
COMM ARCOF
COMM SMOVL C00445 BC00445 V=800.0  +MOVJ EC00445
COMM SMOVL C00446 BC00446 V=1000.0  +MOVJ EC00446
COMM SFTOF3D
COMM 'EndPath W4282
COMM MOVJ C00447 BC00447 VJ=100.00  +MOVJ EC00447 VJ=100.00
COMM MOVJ C00448 BC00448 VJ=100.00  +MOVJ EC00448 VJ=100.00
COMM MOVJ C00449 BC00449 VJ=100.00  +MOVJ EC00449 VJ=100.00
COMM 'Path W4283
COMM SFTOF3D
COMM SFTON3D P022
COMM MOVJ C00450 BC00450 VJ=100.00  +MOVJ EC00450 VJ=100.00
COMM SMOVL C00451 BC00451 V=800.0  +MOVJ EC00451
COMM SMOVL C00452 BC00452 V=150.0 PL=0  +MOVJ EC00452
COMM ARCON
COMM SMOVL C00453 BC00453 V=10.0  +MOVJ EC00453
COMM SMOVL C00454 BC00454 V=10.0  +MOVJ EC00454
COMM SMOVL C00455 BC00455 V=10.0  +MOVJ EC00455
COMM SMOVL C00456 BC00456 V=10.0  +MOVJ EC00456
COMM SMOVL C00457 BC00457 V=10.0  +MOVJ EC00457
COMM SMOVL C00458 BC00458 V=10.0  +MOVJ EC00458
COMM ARCOF
COMM SMOVL C00459 BC00459 V=800.0  +MOVJ EC00459
COMM SMOVL C00460 BC00460 V=1000.0  +MOVJ EC00460
COMM SFTOF3D
COMM 'EndPath W4283
COMM 'Path W4284
COMM SFTOF3D
COMM SFTON3D P024
COMM MOVJ C00461 BC00461 VJ=100.00  +MOVJ EC00461 VJ=100.00
COMM SMOVL C00462 BC00462 V=800.0  +MOVJ EC00462
COMM SMOVL C00463 BC00463 V=150.0 PL=0  +MOVJ EC00463
COMM ARCON
COMM SMOVL C00464 BC00464 V=10.0  +MOVJ EC00464
COMM SMOVL C00465 BC00465 V=10.0  +MOVJ EC00465
COMM SMOVL C00466 BC00466 V=10.0  +MOVJ EC00466
COMM SMOVL C00467 BC00467 V=10.0  +MOVJ EC00467
COMM SMOVL C00468 BC00468 V=10.0  +MOVJ EC00468
COMM SMOVL C00469 BC00469 V=10.0  +MOVJ EC00469
COMM ARCOF
COMM SMOVL C00470 BC00470 V=800.0  +MOVJ EC00470
COMM SMOVL C00471 BC00471 V=1000.0  +MOVJ EC00471
COMM SFTOF3D
COMM 'EndPath W4284
COMM '
COMM MOVJ C00472 BC00472 VJ=100.00  +MOVJ EC00472 VJ=100.00
COMM MOVJ C00473 BC00473 VJ=100.00  +MOVJ EC00473 VJ=100.00
COMM MOVJ C00474 BC00474 VJ=100.00  +MOVJ EC00474 VJ=100.00
COMM 'obrot
COMM MOVJ C00475 BC00475 VJ=100.00  +MOVJ EC00475 VJ=100.00
COMM MOVJ C00476 BC00476 VJ=100.00  +MOVJ EC00476 VJ=100.00
COMM '
'
MOVJ C00477 BC00477 VJ=50.00  +MOVJ EC00477 VJ=50.00
END
